Yaskawa INFORM job: DEMO_ROOF_SIDE_0625_3PAINT_31.JBI

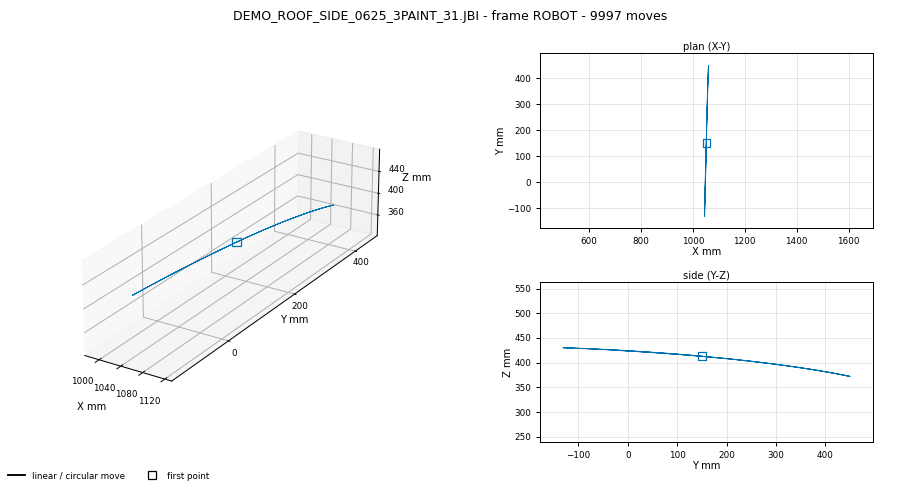
[picture p0: tool path of DEMO_ROOF_SIDE_0625_3PAINT_31.JBI in frame ROBOT, 9997 of 9997 moves have a stored position in this frame; points joined in program order, loops and branches not executed]
/JOB
//NAME DEMO_ROOF_SIDE_0625_3PAINT31
//POS
///NPOS 9997,0,0,0,0,0
///TOOL 0
///USER 0
///POSTYPE ROBOT
///RECTAN
///RCONF 1,0,0,0,0,0,0,0,0,0,0,0,0,0,0,0,0,0,0,0,0,0,0,0
C00000=1052.592,150.571,413.332,171.366,34.299,156.430
C00001=1052.586,150.322,413.353,171.364,34.297,156.430
C00002=1052.580,150.074,413.375,171.362,34.294,156.429
C00003=1052.574,149.824,413.397,171.360,34.291,156.429
C00004=1052.568,149.575,413.419,171.358,34.290,156.428
C00005=1052.563,149.326,413.440,171.357,34.287,156.428
C00006=1052.557,149.077,413.462,171.355,34.285,156.427
C00007=1052.550,148.828,413.484,171.353,34.283,156.427
C00008=1052.544,148.579,413.506,171.351,34.280,156.427
C00009=1052.538,148.331,413.527,171.349,34.278,156.426
C00010=1052.532,148.082,413.549,171.347,34.276,156.426
C00011=1052.526,147.832,413.571,171.345,34.273,156.425
C00012=1052.520,147.583,413.592,171.343,34.271,156.425
C00013=1052.515,147.334,413.614,171.341,34.269,156.425
C00014=1052.508,147.085,413.635,171.339,34.267,156.424
C00015=1052.502,146.836,413.657,171.337,34.264,156.424
C00016=1052.496,146.587,413.678,171.335,34.262,156.424
C00017=1052.490,146.339,413.700,171.334,34.260,156.423
C00018=1052.484,146.089,413.721,171.332,34.258,156.423
C00019=1052.478,145.840,413.743,171.330,34.255,156.422
C00020=1052.472,145.591,413.764,171.328,34.253,156.422
C00021=1052.466,145.342,413.786,171.326,34.251,156.422
C00022=1052.460,145.093,413.807,171.324,34.248,156.421
C00023=1052.454,144.844,413.829,171.322,34.246,156.421
C00024=1052.448,144.595,413.850,171.320,34.244,156.420
C00025=1052.442,144.346,413.872,171.318,34.242,156.420
C00026=1052.436,144.097,413.894,171.316,34.239,156.420
C00027=1052.431,143.849,413.915,171.314,34.237,156.419
C00028=1052.424,143.599,413.936,171.313,34.235,156.419
C00029=1052.418,143.350,413.958,171.311,34.233,156.418
C00030=1052.412,143.101,413.980,171.309,34.230,156.418
C00031=1052.406,142.852,414.001,171.307,34.228,156.418
C00032=1052.400,142.603,414.021,171.305,34.226,156.417
C00033=1052.393,142.318,414.046,171.303,34.223,156.417
C00034=1052.387,142.033,414.071,171.301,34.221,156.416
C00035=1052.380,141.747,414.095,171.298,34.218,156.416
C00036=1052.373,141.462,414.120,171.296,34.216,156.415
C00037=1052.367,141.213,414.142,171.294,34.213,156.415
C00038=1052.361,140.964,414.163,171.292,34.211,156.415
C00039=1052.356,140.715,414.184,171.291,34.209,156.414
C00040=1052.349,140.466,414.205,171.289,34.206,156.414
C00041=1052.343,140.217,414.226,171.287,34.204,156.413
C00042=1052.337,139.968,414.248,171.285,34.202,156.413
C00043=1052.331,139.719,414.269,171.284,34.200,156.413
C00044=1052.325,139.470,414.290,171.282,34.197,156.412
C00045=1052.319,139.221,414.311,171.280,34.195,156.412
C00046=1052.312,138.972,414.333,171.278,34.193,156.411
C00047=1052.307,138.723,414.354,171.275,34.191,156.411
C00048=1052.301,138.473,414.375,171.274,34.189,156.411
C00049=1052.295,138.225,414.396,171.272,34.187,156.410
C00050=1052.289,137.976,414.417,171.270,34.184,156.410
C00051=1052.282,137.727,414.439,171.268,34.182,156.410
C00052=1052.277,137.478,414.459,171.266,34.180,156.409
C00053=1052.271,137.228,414.481,171.265,34.178,156.409
C00054=1052.265,136.980,414.502,171.263,34.175,156.408
C00055=1052.259,136.730,414.522,171.261,34.173,156.408
C00056=1052.253,136.481,414.544,171.259,34.171,156.408
C00057=1052.246,136.233,414.565,171.258,34.169,156.407
C00058=1052.240,135.983,414.586,171.256,34.166,156.407
C00059=1052.235,135.735,414.607,171.254,34.164,156.406
C00060=1052.228,135.485,414.627,171.251,34.162,156.406
C00061=1052.222,135.236,414.649,171.249,34.160,156.406
C00062=1052.217,134.988,414.670,171.248,34.158,156.405
C00063=1052.210,134.738,414.691,171.246,34.155,156.405
C00064=1052.204,134.489,414.712,171.244,34.153,156.405
C00065=1052.199,134.240,414.733,171.242,34.151,156.404
C00066=1052.192,133.991,414.753,171.241,34.149,156.404
C00067=1052.186,133.742,414.774,171.239,34.146,156.403
C00068=1052.181,133.493,414.796,171.237,34.144,156.403
C00069=1052.174,133.244,414.817,171.235,34.142,156.403
C00070=1052.169,132.995,414.837,171.234,34.140,156.402
C00071=1052.163,132.746,414.859,171.232,34.137,156.402
C00072=1052.157,132.497,414.879,171.230,34.136,156.401
C00073=1052.150,132.248,414.900,171.227,34.133,156.401
C00074=1052.145,131.999,414.921,171.226,34.131,156.401
C00075=1052.138,131.750,414.942,171.224,34.129,156.400
C00076=1052.133,131.501,414.963,171.222,34.127,156.400
C00077=1052.126,131.251,414.983,171.220,34.125,156.400
C00078=1052.120,131.002,415.004,171.219,34.122,156.399
C00079=1052.114,130.753,415.024,171.217,34.120,156.399
C00080=1052.108,130.504,415.046,171.215,34.118,156.398
C00081=1052.102,130.255,415.066,171.213,34.116,156.398
C00082=1052.095,130.006,415.086,171.211,34.114,156.398
C00083=1052.090,129.757,415.108,171.210,34.111,156.397
C00084=1052.083,129.508,415.128,171.208,34.109,156.397
C00085=1052.077,129.259,415.149,171.206,34.107,156.397
C00086=1052.071,129.010,415.170,171.204,34.105,156.396
C00087=1052.065,128.761,415.190,171.203,34.103,156.396
C00088=1052.059,128.512,415.211,171.200,34.101,156.395
C00089=1052.053,128.263,415.231,171.198,34.098,156.395
C00090=1052.046,128.013,415.251,171.196,34.096,156.395
C00091=1052.041,127.765,415.273,171.195,34.095,156.394
C00092=1052.034,127.515,415.293,171.193,34.092,156.394
C00093=1052.028,127.266,415.313,171.191,34.090,156.394
C00094=1052.022,127.017,415.334,171.189,34.088,156.393
C00095=1052.016,126.768,415.355,171.188,34.086,156.393
C00096=1052.010,126.519,415.375,171.186,34.084,156.392
C00097=1052.003,126.234,415.399,171.184,34.081,156.392
C00098=1051.996,125.948,415.422,171.182,34.079,156.392
C00099=1051.988,125.663,415.446,171.180,34.076,156.391
C00100=1051.982,125.377,415.469,171.178,34.073,156.391
C00101=1051.975,125.129,415.489,171.176,34.071,156.390
C00102=1051.970,124.879,415.510,171.174,34.070,156.390
C00103=1051.964,124.630,415.530,171.172,34.067,156.390
C00104=1051.958,124.381,415.550,171.170,34.065,156.389
C00105=1051.952,124.131,415.571,171.168,34.063,156.389
C00106=1051.945,123.883,415.592,171.167,34.061,156.388
C00107=1051.939,123.634,415.612,171.165,34.059,156.388
C00108=1051.934,123.384,415.633,171.163,34.056,156.388
C00109=1051.928,123.136,415.653,171.162,34.054,156.387
C00110=1051.921,122.886,415.673,171.160,34.052,156.387
C00111=1051.916,122.637,415.694,171.158,34.050,156.387
C00112=1051.909,122.387,415.714,171.156,34.048,156.386
C00113=1051.903,122.139,415.735,171.155,34.046,156.386
C00114=1051.898,121.890,415.755,171.153,34.043,156.386
C00115=1051.891,121.641,415.776,171.151,34.041,156.385
C00116=1051.885,121.392,415.795,171.150,34.039,156.385
C00117=1051.880,121.143,415.816,171.147,34.037,156.384
C00118=1051.873,120.893,415.836,171.145,34.035,156.384
C00119=1051.867,120.644,415.856,171.143,34.032,156.384
C00120=1051.861,120.396,415.876,171.142,34.031,156.383
C00121=1051.855,120.146,415.897,171.140,34.028,156.383
C00122=1051.849,119.897,415.917,171.138,34.026,156.383
C00123=1051.843,119.648,415.937,171.137,34.024,156.382
C00124=1051.838,119.398,415.958,171.135,34.022,156.382
C00125=1051.832,119.149,415.978,171.133,34.020,156.381
C00126=1051.825,118.901,415.999,171.132,34.017,156.381
C00127=1051.819,118.652,416.019,171.130,34.015,156.381
C00128=1051.813,118.403,416.040,171.128,34.013,156.380
C00129=1051.807,118.154,416.059,171.126,34.011,156.380
C00130=1051.801,117.904,416.080,171.125,34.009,156.380
C00131=1051.796,117.655,416.100,171.123,34.006,156.379
C00132=1051.790,117.406,416.120,171.121,34.004,156.379
C00133=1051.784,117.157,416.140,171.119,34.002,156.378
C00134=1051.777,116.907,416.160,171.117,34.000,156.378
C00135=1051.772,116.658,416.180,171.115,33.998,156.378
C00136=1051.766,116.409,416.200,171.114,33.995,156.377
C00137=1051.760,116.161,416.220,171.112,33.993,156.377
C00138=1051.753,115.911,416.241,171.110,33.991,156.376
C00139=1051.748,115.662,416.261,171.109,33.989,156.376
C00140=1051.742,115.413,416.281,171.107,33.987,156.376
C00141=1051.736,115.164,416.301,171.105,33.984,156.375
C00142=1051.730,114.915,416.321,171.104,33.982,156.375
C00143=1051.724,114.666,416.342,171.102,33.980,156.375
C00144=1051.718,114.417,416.362,171.100,33.978,156.374
C00145=1051.713,114.168,416.381,171.099,33.975,156.374
C00146=1051.706,113.918,416.402,171.097,33.973,156.374
C00147=1051.700,113.669,416.422,171.095,33.971,156.373
C00148=1051.695,113.420,416.442,171.094,33.969,156.373
C00149=1051.689,113.171,416.462,171.092,33.967,156.372
C00150=1051.683,112.921,416.482,171.089,33.965,156.372
C00151=1051.677,112.672,416.502,171.088,33.963,156.372
C00152=1051.671,112.424,416.522,171.086,33.961,156.371
C00153=1051.665,112.175,416.542,171.084,33.959,156.371
C00154=1051.658,111.925,416.561,171.083,33.956,156.371
C00155=1051.652,111.676,416.581,171.081,33.954,156.370
C00156=1051.646,111.427,416.601,171.079,33.952,156.370
C00157=1051.640,111.178,416.621,171.078,33.950,156.369
C00158=1051.634,110.928,416.641,171.076,33.948,156.369
C00159=1051.627,110.679,416.660,171.074,33.946,156.369
C00160=1051.621,110.431,416.680,171.072,33.944,156.368
C00161=1051.615,110.145,416.703,171.071,33.941,156.368
C00162=1051.607,109.859,416.725,171.069,33.939,156.368
C00163=1051.601,109.574,416.748,171.067,33.936,156.367
C00164=1051.594,109.288,416.770,171.065,33.934,156.367
C00165=1051.588,109.039,416.790,171.063,33.932,156.366
C00166=1051.581,108.790,416.810,171.061,33.930,156.366
C00167=1051.575,108.540,416.830,171.059,33.928,156.366
C00168=1051.569,108.292,416.849,171.057,33.926,156.365
C00169=1051.563,108.042,416.868,171.055,33.923,156.365
C00170=1051.557,107.793,416.888,171.054,33.921,156.365
C00171=1051.550,107.544,416.909,171.052,33.919,156.364
C00172=1051.545,107.294,416.928,171.050,33.917,156.364
C00173=1051.539,107.046,416.948,171.049,33.915,156.364
C00174=1051.532,106.797,416.966,171.047,33.913,156.363
C00175=1051.526,106.548,416.986,171.045,33.911,156.363
C00176=1051.520,106.298,417.007,171.044,33.908,156.362
C00177=1051.514,106.049,417.026,171.042,33.906,156.362
C00178=1051.508,105.800,417.046,171.040,33.905,156.362
C00179=1051.502,105.551,417.065,171.039,33.903,156.361
C00180=1051.495,105.302,417.085,171.037,33.900,156.361
C00181=1051.490,105.053,417.104,171.035,33.898,156.361
C00182=1051.484,104.804,417.124,171.034,33.896,156.360
C00183=1051.478,104.554,417.143,171.032,33.894,156.360
C00184=1051.472,104.305,417.163,171.030,33.892,156.360
C00185=1051.466,104.055,417.183,171.029,33.890,156.359
C00186=1051.459,103.807,417.202,171.027,33.888,156.359
C00187=1051.453,103.557,417.221,171.025,33.885,156.359
C00188=1051.447,103.309,417.241,171.023,33.883,156.358
C00189=1051.442,103.059,417.260,171.021,33.881,156.358
C00190=1051.436,102.810,417.280,171.020,33.879,156.357
C00191=1051.429,102.561,417.299,171.018,33.877,156.357
C00192=1051.423,102.311,417.319,171.016,33.875,156.357
C00193=1051.417,102.062,417.339,171.015,33.872,156.356
C00194=1051.411,101.813,417.358,171.013,33.870,156.356
C00195=1051.405,101.564,417.378,171.011,33.868,156.356
C00196=1051.399,101.315,417.396,171.010,33.866,156.355
C00197=1051.393,101.066,417.416,171.008,33.864,156.355
C00198=1051.387,100.817,417.436,171.006,33.862,156.355
C00199=1051.382,100.567,417.455,171.005,33.860,156.354
C00200=1051.375,100.318,417.473,171.003,33.857,156.354
C00201=1051.369,100.069,417.493,171.001,33.856,156.353
C00202=1051.363,99.820,417.512,171.000,33.854,156.353
C00203=1051.356,99.570,417.532,170.998,33.852,156.353
C00204=1051.350,99.321,417.552,170.996,33.850,156.353
C00205=1051.344,99.072,417.570,170.995,33.847,156.352
C00206=1051.338,98.823,417.590,170.993,33.845,156.352
C00207=1051.332,98.574,417.609,170.991,33.843,156.351
C00208=1051.326,98.325,417.628,170.989,33.841,156.351
C00209=1051.319,98.076,417.647,170.987,33.839,156.351
C00210=1051.314,97.826,417.666,170.986,33.837,156.350
C00211=1051.307,97.578,417.685,170.984,33.835,156.350
C00212=1051.301,97.328,417.705,170.982,33.833,156.350
C00213=1051.296,97.079,417.724,170.981,33.831,156.349
C00214=1051.289,96.830,417.743,170.979,33.829,156.349
C00215=1051.284,96.580,417.762,170.977,33.826,156.349
C00216=1051.277,96.332,417.781,170.976,33.825,156.348
C00217=1051.271,96.082,417.801,170.974,33.823,156.348
C00218=1051.264,95.833,417.819,170.972,33.821,156.348
C00219=1051.258,95.583,417.839,170.971,33.818,156.347
C00220=1051.252,95.334,417.857,170.969,33.816,156.347
C00221=1051.246,95.085,417.877,170.968,33.814,156.347
C00222=1051.240,94.836,417.896,170.966,33.812,156.346
C00223=1051.234,94.587,417.915,170.964,33.810,156.346
C00224=1051.227,94.338,417.934,170.963,33.808,156.345
C00225=1051.221,94.053,417.956,170.961,33.806,156.345
C00226=1051.213,93.766,417.977,170.959,33.803,156.345
C00227=1051.207,93.481,417.999,170.957,33.801,156.344
C00228=1051.200,93.196,418.021,170.954,33.798,156.344
C00229=1051.194,92.946,418.040,170.953,33.796,156.343
C00230=1051.188,92.697,418.059,170.951,33.794,156.343
C00231=1051.182,92.448,418.078,170.949,33.792,156.343
C00232=1051.176,92.199,418.097,170.948,33.790,156.342
C00233=1051.170,91.950,418.116,170.946,33.788,156.342
C00234=1051.163,91.701,418.135,170.944,33.786,156.342
C00235=1051.158,91.451,418.154,170.943,33.784,156.341
C00236=1051.151,91.202,418.173,170.941,33.781,156.341
C00237=1051.146,90.953,418.192,170.939,33.779,156.341
C00238=1051.140,90.703,418.211,170.938,33.777,156.340
C00239=1051.134,90.454,418.230,170.936,33.775,156.340
C00240=1051.127,90.205,418.249,170.935,33.773,156.340
C00241=1051.121,89.955,418.268,170.933,33.771,156.339
C00242=1051.115,89.706,418.287,170.931,33.769,156.339
C00243=1051.109,89.457,418.305,170.930,33.767,156.339
C00244=1051.102,89.208,418.324,170.928,33.765,156.338
C00245=1051.096,88.959,418.343,170.926,33.763,156.338
C00246=1051.090,88.710,418.362,170.925,33.761,156.338
C00247=1051.084,88.460,418.380,170.923,33.759,156.337
C00248=1051.077,88.211,418.398,170.921,33.756,156.337
C00249=1051.072,87.961,418.418,170.920,33.755,156.337
C00250=1051.065,87.712,418.436,170.918,33.753,156.336
C00251=1051.059,87.463,418.455,170.917,33.751,156.336
C00252=1051.053,87.215,418.473,170.915,33.749,156.336
C00253=1051.047,86.965,418.492,170.913,33.747,156.335
C00254=1051.041,86.716,418.511,170.911,33.745,156.335
C00255=1051.035,86.467,418.530,170.909,33.742,156.335
C00256=1051.028,86.217,418.548,170.907,33.740,156.334
C00257=1051.022,85.968,418.566,170.906,33.738,156.334
C00258=1051.016,85.719,418.586,170.904,33.736,156.334
C00259=1051.010,85.469,418.604,170.903,33.734,156.333
C00260=1051.004,85.220,418.623,170.901,33.732,156.333
C00261=1050.997,84.971,418.641,170.899,33.730,156.333
C00262=1050.992,84.721,418.660,170.898,33.728,156.332
C00263=1050.986,84.473,418.678,170.896,33.726,156.332
C00264=1050.979,84.224,418.697,170.894,33.724,156.331
C00265=1050.973,83.975,418.716,170.893,33.722,156.331
C00266=1050.967,83.725,418.734,170.891,33.720,156.331
C00267=1050.961,83.475,418.753,170.890,33.718,156.331
C00268=1050.955,83.226,418.771,170.888,33.716,156.330
C00269=1050.948,82.977,418.790,170.886,33.714,156.330
C00270=1050.943,82.729,418.808,170.885,33.712,156.329
C00271=1050.937,82.479,418.827,170.883,33.710,156.329
C00272=1050.931,82.230,418.846,170.881,33.708,156.329
C00273=1050.924,81.980,418.864,170.880,33.705,156.328
C00274=1050.918,81.731,418.882,170.878,33.703,156.328
C00275=1050.912,81.482,418.901,170.877,33.701,156.328
C00276=1050.907,81.233,418.920,170.875,33.699,156.327
C00277=1050.900,80.984,418.938,170.873,33.697,156.327
C00278=1050.894,80.734,418.956,170.872,33.695,156.327
C00279=1050.888,80.485,418.975,170.870,33.693,156.326
C00280=1050.881,80.236,418.994,170.868,33.691,156.326
C00281=1050.876,79.987,419.011,170.866,33.689,156.326
C00282=1050.870,79.737,419.030,170.864,33.687,156.325
C00283=1050.864,79.488,419.049,170.863,33.685,156.325
C00284=1050.858,79.238,419.067,170.861,33.682,156.325
C00285=1050.851,78.989,419.086,170.859,33.680,156.324
C00286=1050.846,78.740,419.103,170.858,33.679,156.324
C00287=1050.839,78.491,419.122,170.856,33.677,156.324
C00288=1050.833,78.242,419.140,170.855,33.675,156.323
C00289=1050.826,77.956,419.162,170.853,33.672,156.323
C00290=1050.819,77.670,419.182,170.851,33.670,156.323
C00291=1050.812,77.384,419.203,170.849,33.667,156.322
C00292=1050.805,77.099,419.224,170.847,33.665,156.322
C00293=1050.798,76.850,419.243,170.845,33.663,156.321
C00294=1050.793,76.601,419.260,170.844,33.661,156.321
C00295=1050.786,76.352,419.279,170.842,33.659,156.321
C00296=1050.780,76.102,419.297,170.841,33.657,156.320
C00297=1050.774,75.853,419.315,170.839,33.655,156.320
C00298=1050.768,75.603,419.333,170.837,33.653,156.320
C00299=1050.762,75.354,419.352,170.836,33.651,156.319
C00300=1050.756,75.105,419.370,170.834,33.649,156.319
C00301=1050.749,74.856,419.388,170.832,33.647,156.319
C00302=1050.743,74.606,419.406,170.831,33.645,156.318
C00303=1050.737,74.357,419.424,170.829,33.643,156.318
C00304=1050.731,74.108,419.442,170.828,33.641,156.318
C00305=1050.725,73.859,419.461,170.826,33.639,156.317
C00306=1050.718,73.609,419.478,170.824,33.637,156.317
C00307=1050.713,73.360,419.496,170.823,33.635,156.317
C00308=1050.706,73.111,419.515,170.821,33.633,156.316
C00309=1050.700,72.861,419.532,170.820,33.631,156.316
C00310=1050.694,72.612,419.551,170.818,33.629,156.316
C00311=1050.688,72.363,419.569,170.816,33.626,156.315
C00312=1050.682,72.113,419.587,170.814,33.624,156.315
C00313=1050.676,71.864,419.605,170.812,33.622,156.315
C00314=1050.670,71.615,419.623,170.810,33.620,156.314
C00315=1050.664,71.366,419.641,170.809,33.619,156.314
C00316=1050.657,71.117,419.659,170.807,33.617,156.314
C00317=1050.651,70.867,419.677,170.806,33.615,156.313
C00318=1050.645,70.618,419.695,170.804,33.613,156.313
C00319=1050.639,70.369,419.713,170.802,33.611,156.313
C00320=1050.633,70.119,419.731,170.801,33.608,156.312
C00321=1050.627,69.871,419.749,170.799,33.606,156.312
C00322=1050.621,69.621,419.767,170.797,33.604,156.312
C00323=1050.614,69.371,419.784,170.796,33.602,156.311
C00324=1050.608,69.122,419.802,170.794,33.600,156.311
C00325=1050.602,68.873,419.821,170.793,33.598,156.311
C00326=1050.596,68.623,419.839,170.791,33.596,156.310
C00327=1050.590,68.374,419.856,170.789,33.594,156.310
C00328=1050.583,68.125,419.874,170.788,33.592,156.310
C00329=1050.577,67.876,419.892,170.786,33.590,156.309
C00330=1050.571,67.627,419.910,170.784,33.588,156.309
C00331=1050.565,67.377,419.928,170.783,33.586,156.309
C00332=1050.558,67.128,419.945,170.781,33.584,156.309
C00333=1050.553,66.879,419.963,170.780,33.582,156.308
C00334=1050.546,66.630,419.981,170.778,33.580,156.308
C00335=1050.540,66.380,419.999,170.776,33.578,156.307
C00336=1050.534,66.131,420.016,170.775,33.576,156.307
C00337=1050.528,65.881,420.034,170.773,33.574,156.307
C00338=1050.521,65.632,420.051,170.771,33.572,156.306
C00339=1050.515,65.383,420.070,170.770,33.570,156.306
C00340=1050.509,65.134,420.088,170.768,33.568,156.306
C00341=1050.503,64.884,420.106,170.767,33.566,156.306
C00342=1050.497,64.635,420.123,170.765,33.564,156.305
C00343=1050.491,64.386,420.140,170.763,33.562,156.305
C00344=1050.485,64.136,420.158,170.762,33.560,156.305
C00345=1050.478,63.887,420.175,170.760,33.558,156.304
C00346=1050.472,63.637,420.193,170.758,33.556,156.304
C00347=1050.466,63.389,420.210,170.757,33.554,156.304
C00348=1050.459,63.140,420.228,170.755,33.552,156.303
C00349=1050.453,62.890,420.246,170.753,33.550,156.303
C00350=1050.446,62.641,420.263,170.752,33.548,156.303
C00351=1050.440,62.392,420.281,170.750,33.546,156.302
C00352=1050.433,62.142,420.298,170.749,33.545,156.302
C00353=1050.426,61.856,420.318,170.746,33.543,156.302
C00354=1050.419,61.570,420.338,170.744,33.541,156.301
C00355=1050.412,61.284,420.358,170.742,33.538,156.301
C00356=1050.405,60.999,420.378,170.740,33.536,156.301
C00357=1050.399,60.749,420.396,170.738,33.534,156.300
C00358=1050.392,60.500,420.413,170.737,33.532,156.300
C00359=1050.386,60.251,420.431,170.735,33.530,156.300
C00360=1050.379,60.001,420.448,170.733,33.528,156.299
C00361=1050.374,59.752,420.465,170.732,33.526,156.299
C00362=1050.367,59.503,420.483,170.730,33.524,156.299
C00363=1050.361,59.254,420.500,170.729,33.522,156.298
C00364=1050.355,59.004,420.518,170.727,33.520,156.298
C00365=1050.348,58.755,420.535,170.725,33.518,156.298
C00366=1050.342,58.506,420.553,170.724,33.516,156.297
C00367=1050.335,58.256,420.570,170.722,33.514,156.297
C00368=1050.329,58.008,420.587,170.720,33.513,156.297
C00369=1050.323,57.758,420.605,170.719,33.511,156.297
C00370=1050.317,57.509,420.622,170.717,33.509,156.296
C00371=1050.311,57.259,420.639,170.715,33.507,156.296
C00372=1050.305,57.010,420.656,170.714,33.505,156.296
C00373=1050.298,56.761,420.673,170.712,33.503,156.295
C00374=1050.292,56.511,420.691,170.711,33.501,156.295
C00375=1050.285,56.262,420.708,170.709,33.499,156.295
C00376=1050.279,56.012,420.726,170.707,33.497,156.294
C00377=1050.273,55.763,420.742,170.706,33.495,156.294
C00378=1050.267,55.514,420.760,170.704,33.493,156.294
C00379=1050.261,55.264,420.777,170.702,33.491,156.293
C00380=1050.254,55.015,420.795,170.701,33.489,156.293
C00381=1050.249,54.766,420.812,170.699,33.487,156.293
C00382=1050.242,54.516,420.829,170.697,33.485,156.293
C00383=1050.236,54.267,420.846,170.696,33.483,156.292
C00384=1050.230,54.017,420.864,170.694,33.481,156.292
C00385=1050.223,53.769,420.881,170.692,33.479,156.292
C00386=1050.217,53.519,420.898,170.691,33.477,156.291
C00387=1050.211,53.270,420.915,170.689,33.475,156.291
C00388=1050.205,53.020,420.932,170.688,33.473,156.291
C00389=1050.199,52.771,420.950,170.686,33.471,156.290
C00390=1050.193,52.522,420.967,170.684,33.469,156.290
C00391=1050.186,52.272,420.983,170.683,33.467,156.290
C00392=1050.181,52.023,421.001,170.681,33.465,156.289
C00393=1050.174,51.774,421.018,170.679,33.463,156.289
C00394=1050.168,51.525,421.035,170.678,33.462,156.289
C00395=1050.162,51.275,421.053,170.676,33.459,156.288
C00396=1050.155,51.026,421.069,170.674,33.457,156.288
C00397=1050.149,50.776,421.086,170.673,33.456,156.288
C00398=1050.143,50.527,421.104,170.671,33.454,156.287
C00399=1050.137,50.278,421.121,170.670,33.452,156.287
C00400=1050.131,50.028,421.137,170.668,33.450,156.287
C00401=1050.125,49.779,421.155,170.666,33.448,156.287
C00402=1050.118,49.530,421.172,170.665,33.446,156.286
C00403=1050.113,49.280,421.189,170.663,33.444,156.286
C00404=1050.107,49.031,421.206,170.661,33.442,156.286
C00405=1050.100,48.782,421.223,170.660,33.440,156.285
C00406=1050.095,48.532,421.240,170.658,33.438,156.285
C00407=1050.088,48.283,421.258,170.657,33.436,156.285
C00408=1050.082,48.034,421.274,170.655,33.434,156.284
C00409=1050.076,47.785,421.291,170.653,33.432,156.284
C00410=1050.069,47.535,421.309,170.652,33.430,156.284
C00411=1050.064,47.286,421.325,170.650,33.428,156.283
C00412=1050.057,47.037,421.342,170.648,33.426,156.283
C00413=1050.051,46.787,421.359,170.647,33.424,156.283
C00414=1050.045,46.538,421.376,170.644,33.422,156.282
C00415=1050.039,46.289,421.392,170.642,33.420,156.282
C00416=1050.033,46.039,421.410,170.641,33.418,156.282
C00417=1050.026,45.752,421.430,170.639,33.415,156.281
C00418=1050.019,45.467,421.449,170.637,33.413,156.281
C00419=1050.012,45.180,421.468,170.635,33.411,156.281
C00420=1050.005,44.894,421.488,170.633,33.409,156.280
C00421=1049.999,44.645,421.504,170.632,33.407,156.280
C00422=1049.993,44.396,421.521,170.630,33.405,156.280
C00423=1049.988,44.146,421.538,170.628,33.403,156.279
C00424=1049.981,43.897,421.555,170.627,33.401,156.279
C00425=1049.975,43.648,421.572,170.625,33.399,156.279
C00426=1049.969,43.399,421.589,170.623,33.397,156.278
C00427=1049.963,43.149,421.606,170.622,33.395,156.278
C00428=1049.957,42.900,421.623,170.620,33.393,156.278
C00429=1049.951,42.650,421.639,170.619,33.391,156.277
C00430=1049.944,42.400,421.656,170.617,33.389,156.277
C00431=1049.938,42.152,421.673,170.615,33.387,156.277
C00432=1049.932,41.902,421.689,170.614,33.386,156.277
C00433=1049.925,41.652,421.706,170.612,33.384,156.276
C00434=1049.919,41.404,421.723,170.610,33.382,156.276
C00435=1049.913,41.154,421.739,170.609,33.380,156.276
C00436=1049.906,40.905,421.756,170.607,33.378,156.275
C00437=1049.900,40.655,421.772,170.605,33.376,156.275
C00438=1049.894,40.406,421.789,170.604,33.374,156.275
C00439=1049.888,40.157,421.806,170.602,33.372,156.274
C00440=1049.882,39.907,421.822,170.600,33.370,156.274
C00441=1049.876,39.658,421.839,170.599,33.368,156.274
C00442=1049.870,39.409,421.855,170.597,33.366,156.273
C00443=1049.863,39.159,421.872,170.595,33.364,156.273
C00444=1049.858,38.910,421.889,170.594,33.362,156.273
C00445=1049.852,38.660,421.905,170.592,33.360,156.273
C00446=1049.845,38.411,421.922,170.590,33.358,156.272
C00447=1049.839,38.161,421.939,170.589,33.356,156.272
C00448=1049.833,37.912,421.955,170.587,33.354,156.272
C00449=1049.827,37.663,421.971,170.585,33.352,156.271
C00450=1049.821,37.414,421.988,170.584,33.350,156.271
C00451=1049.813,37.164,422.004,170.582,33.348,156.271
C00452=1049.807,36.915,422.021,170.580,33.347,156.271
C00453=1049.801,36.666,422.037,170.579,33.345,156.270
C00454=1049.795,36.415,422.054,170.577,33.343,156.270
C00455=1049.789,36.166,422.070,170.575,33.341,156.270
C00456=1049.783,35.917,422.087,170.574,33.339,156.269
C00457=1049.777,35.668,422.103,170.572,33.338,156.269
C00458=1049.769,35.418,422.119,170.570,33.336,156.269
C00459=1049.764,35.169,422.135,170.569,33.334,156.268
C00460=1049.758,34.920,422.152,170.567,33.332,156.268
C00461=1049.752,34.670,422.168,170.565,33.330,156.268
C00462=1049.745,34.421,422.185,170.564,33.328,156.268
C00463=1049.739,34.171,422.201,170.562,33.326,156.267
C00464=1049.732,33.922,422.217,170.560,33.324,156.267
C00465=1049.726,33.673,422.233,170.558,33.322,156.267
C00466=1049.720,33.424,422.250,170.557,33.320,156.266
C00467=1049.714,33.174,422.266,170.555,33.318,156.266
C00468=1049.708,32.924,422.282,170.553,33.317,156.266
C00469=1049.701,32.675,422.298,170.552,33.315,156.266
C00470=1049.695,32.426,422.314,170.550,33.313,156.265
C00471=1049.689,32.177,422.331,170.548,33.311,156.265
C00472=1049.683,31.927,422.347,170.547,33.309,156.265
C00473=1049.677,31.677,422.364,170.545,33.307,156.264
C00474=1049.671,31.428,422.380,170.543,33.306,156.264
C00475=1049.664,31.179,422.395,170.542,33.304,156.264
C00476=1049.658,30.929,422.412,170.540,33.302,156.264
C00477=1049.651,30.679,422.428,170.538,33.300,156.263
C00478=1049.646,30.430,422.445,170.537,33.298,156.263
C00479=1049.640,30.181,422.461,170.535,33.296,156.263
C00480=1049.633,29.932,422.476,170.533,33.294,156.262
C00481=1049.625,29.645,422.495,170.531,33.292,156.262
C00482=1049.619,29.360,422.514,170.529,33.290,156.262
C00483=1049.612,29.073,422.533,170.527,33.288,156.261
C00484=1049.605,28.787,422.551,170.526,33.286,156.261
C00485=1049.599,28.538,422.568,170.524,33.284,156.261
C00486=1049.592,28.289,422.583,170.522,33.282,156.260
C00487=1049.586,28.039,422.599,170.520,33.280,156.260
C00488=1049.580,27.790,422.616,170.519,33.278,156.260
C00489=1049.573,27.540,422.631,170.517,33.276,156.260
C00490=1049.567,27.290,422.647,170.515,33.274,156.259
C00491=1049.560,27.041,422.663,170.514,33.272,156.259
C00492=1049.555,26.792,422.679,170.512,33.271,156.259
C00493=1049.549,26.543,422.695,170.510,33.269,156.258
C00494=1049.542,26.294,422.711,170.509,33.267,156.258
C00495=1049.536,26.044,422.727,170.507,33.265,156.258
C00496=1049.530,25.794,422.743,170.505,33.263,156.258
C00497=1049.523,25.545,422.759,170.503,33.261,156.257
C00498=1049.517,25.295,422.775,170.502,33.259,156.257
C00499=1049.510,25.046,422.791,170.500,33.257,156.257
C00500=1049.504,24.797,422.807,170.498,33.256,156.257
C00501=1049.498,24.548,422.823,170.497,33.254,156.256
C00502=1049.492,24.298,422.838,170.495,33.252,156.256
C00503=1049.486,24.048,422.855,170.493,33.251,156.256
C00504=1049.479,23.799,422.870,170.491,33.249,156.255
C00505=1049.473,23.550,422.886,170.490,33.247,156.255
C00506=1049.466,23.300,422.902,170.488,33.245,156.255
C00507=1049.461,23.050,422.918,170.486,33.243,156.255
C00508=1049.454,22.801,422.934,170.485,33.241,156.254
C00509=1049.448,22.552,422.950,170.483,33.239,156.254
C00510=1049.442,22.302,422.965,170.481,33.237,156.254
C00511=1049.436,22.053,422.981,170.480,33.236,156.253
C00512=1049.430,21.804,422.997,170.478,33.234,156.253
C00513=1049.423,21.554,423.012,170.476,33.232,156.253
C00514=1049.417,21.305,423.029,170.474,33.230,156.253
C00515=1049.411,21.056,423.044,170.473,33.228,156.252
C00516=1049.405,20.806,423.060,170.471,33.226,156.252
C00517=1049.398,20.557,423.075,170.469,33.224,156.252
C00518=1049.392,20.307,423.092,170.468,33.223,156.252
C00519=1049.386,20.058,423.107,170.466,33.221,156.251
C00520=1049.380,19.808,423.123,170.464,33.219,156.251
C00521=1049.373,19.559,423.139,170.462,33.218,156.251
C00522=1049.368,19.309,423.154,170.461,33.216,156.250
C00523=1049.361,19.060,423.170,170.459,33.214,156.250
C00524=1049.355,18.811,423.186,170.457,33.212,156.250
C00525=1049.349,18.561,423.201,170.455,33.210,156.250
C00526=1049.342,18.312,423.217,170.454,33.208,156.249
C00527=1049.336,18.062,423.232,170.452,33.207,156.249
C00528=1049.330,17.813,423.248,170.450,33.205,156.249
C00529=1049.324,17.563,423.263,170.449,33.203,156.248
C00530=1049.317,17.314,423.279,170.447,33.201,156.248
C00531=1049.311,17.064,423.294,170.445,33.199,156.248
C00532=1049.305,16.815,423.310,170.443,33.197,156.248
C00533=1049.298,16.566,423.326,170.442,33.196,156.247
C00534=1049.293,16.316,423.341,170.440,33.194,156.247
C00535=1049.286,16.067,423.357,170.438,33.192,156.247
C00536=1049.280,15.817,423.372,170.436,33.191,156.247
C00537=1049.274,15.568,423.388,170.435,33.189,156.246
C00538=1049.267,15.318,423.403,170.433,33.187,156.246
C00539=1049.261,15.069,423.420,170.431,33.185,156.246
C00540=1049.255,14.819,423.435,170.429,33.183,156.246
C00541=1049.248,14.570,423.450,170.428,33.181,156.245
C00542=1049.243,14.320,423.466,170.426,33.180,156.245
C00543=1049.236,14.071,423.481,170.424,33.178,156.245
C00544=1049.229,13.822,423.496,170.422,33.176,156.244
C00545=1049.224,13.605,423.509,170.421,33.174,156.244
C00546=1049.218,13.389,423.523,170.419,33.173,156.244
C00547=1049.213,13.173,423.536,170.418,33.172,156.244
C00548=1049.208,12.957,423.550,170.416,33.170,156.244
C00549=1049.202,12.740,423.563,170.415,33.168,156.243
C00550=1049.196,12.524,423.576,170.413,33.167,156.243
C00551=1049.191,12.307,423.589,170.412,33.166,156.243
C00552=1049.185,12.091,423.603,170.410,33.164,156.243
C00553=1049.179,11.842,423.618,170.408,33.162,156.242
C00554=1049.173,11.592,423.633,170.407,33.161,156.242
C00555=1049.166,11.343,423.648,170.405,33.159,156.242
C00556=1049.160,11.093,423.664,170.403,33.157,156.242
C00557=1049.154,10.843,423.679,170.401,33.155,156.241
C00558=1049.147,10.594,423.694,170.400,33.154,156.241
C00559=1049.141,10.345,423.709,170.398,33.152,156.241
C00560=1049.135,10.096,423.724,170.397,33.150,156.241
C00561=1049.129,9.846,423.739,170.395,33.148,156.240
C00562=1049.122,9.597,423.755,170.394,33.147,156.240
C00563=1049.116,9.347,423.770,170.392,33.145,156.240
C00564=1049.110,9.097,423.785,170.390,33.143,156.240
C00565=1049.103,8.848,423.801,170.388,33.142,156.239
C00566=1049.097,8.599,423.816,170.386,33.140,156.239
C00567=1049.090,8.349,423.831,170.385,33.138,156.239
C00568=1049.084,8.099,423.846,170.383,33.136,156.239
C00569=1049.077,7.850,423.861,170.381,33.135,156.238
C00570=1049.072,7.601,423.876,170.379,33.133,156.238
C00571=1049.066,7.351,423.891,170.378,33.131,156.238
C00572=1049.060,7.102,423.906,170.376,33.129,156.238
C00573=1049.051,6.751,423.928,170.373,33.127,156.237
C00574=1049.042,6.399,423.949,170.371,33.125,156.237
C00575=1049.033,6.049,423.970,170.368,33.122,156.237
C00576=1049.024,5.697,423.991,170.366,33.120,156.236
C00577=1049.018,5.447,424.006,170.364,33.118,156.236
C00578=1049.011,5.198,424.022,170.362,33.116,156.236
C00579=1049.005,4.949,424.037,170.360,33.114,156.235
C00580=1048.999,4.699,424.052,170.359,33.113,156.235
C00581=1048.993,4.450,424.066,170.357,33.111,156.235
C00582=1048.986,4.200,424.081,170.355,33.109,156.235
C00583=1048.980,3.951,424.096,170.353,33.107,156.234
C00584=1048.974,3.701,424.111,170.352,33.106,156.234
C00585=1048.967,3.451,424.126,170.350,33.104,156.234
C00586=1048.961,3.203,424.141,170.348,33.103,156.234
C00587=1048.955,2.953,424.157,170.346,33.101,156.233
C00588=1048.949,2.703,424.172,170.344,33.099,156.233
C00589=1048.943,2.454,424.187,170.343,33.097,156.233
C00590=1048.937,2.205,424.201,170.341,33.096,156.233
C00591=1048.931,1.955,424.216,170.339,33.094,156.232
C00592=1048.924,1.706,424.231,170.337,33.092,156.232
C00593=1048.918,1.456,424.246,170.335,33.090,156.232
C00594=1048.912,1.207,424.261,170.334,33.088,156.232
C00595=1048.906,0.957,424.276,170.332,33.087,156.231
C00596=1048.899,0.708,424.291,170.330,33.085,156.231
C00597=1048.893,0.458,424.306,170.328,33.083,156.231
C00598=1048.887,0.209,424.320,170.326,33.081,156.231
C00599=1048.881,-0.041,424.335,170.325,33.080,156.230
C00600=1048.874,-0.290,424.350,170.323,33.078,156.230
C00601=1048.869,-0.539,424.365,170.321,33.077,156.230
C00602=1048.862,-0.789,424.380,170.319,33.075,156.230
C00603=1048.857,-1.039,424.395,170.317,33.073,156.229
C00604=1048.850,-1.289,424.410,170.316,33.071,156.229
C00605=1048.844,-1.537,424.425,170.314,33.070,156.229
C00606=1048.838,-1.787,424.440,170.312,33.068,156.229
C00607=1048.832,-2.037,424.454,170.310,33.066,156.228
C00608=1048.826,-2.286,424.469,170.308,33.064,156.228
C00609=1048.819,-2.569,424.485,170.306,33.062,156.228
C00610=1048.811,-2.852,424.502,170.304,33.060,156.228
C00611=1048.805,-3.135,424.518,170.302,33.059,156.227
C00612=1048.797,-3.418,424.536,170.300,33.057,156.227
C00613=1048.791,-3.667,424.550,170.298,33.055,156.227
C00614=1048.785,-3.918,424.565,170.297,33.053,156.227
C00615=1048.779,-4.167,424.579,170.295,33.052,156.226
C00616=1048.772,-4.416,424.594,170.293,33.050,156.226
C00617=1048.766,-4.666,424.609,170.291,33.048,156.226
C00618=1048.760,-4.915,424.623,170.289,33.047,156.226
C00619=1048.754,-5.164,424.638,170.287,33.045,156.225
C00620=1048.747,-5.414,424.652,170.286,33.044,156.225
C00621=1048.741,-5.663,424.666,170.284,33.042,156.225
C00622=1048.735,-5.913,424.681,170.283,33.040,156.225
C00623=1048.728,-6.162,424.696,170.281,33.039,156.225
C00624=1048.721,-6.412,424.710,170.279,33.037,156.224
C00625=1048.716,-6.661,424.724,170.277,33.035,156.224
C00626=1048.709,-6.911,424.739,170.276,33.034,156.224
C00627=1048.702,-7.160,424.754,170.274,33.032,156.224
C00628=1048.697,-7.410,424.768,170.272,33.030,156.223
C00629=1048.690,-7.660,424.783,170.270,33.029,156.223
C00630=1048.684,-7.909,424.797,170.268,33.028,156.223
C00631=1048.678,-8.158,424.811,170.266,33.025,156.223
C00632=1048.671,-8.408,424.826,170.264,33.024,156.222
C00633=1048.665,-8.657,424.840,170.263,33.023,156.222
C00634=1048.659,-8.907,424.854,170.261,33.021,156.222
C00635=1048.652,-9.157,424.869,170.259,33.019,156.222
C00636=1048.646,-9.406,424.883,170.257,33.018,156.222
C00637=1048.640,-9.656,424.898,170.255,33.016,156.221
C00638=1048.634,-9.905,424.912,170.253,33.014,156.221
C00639=1048.628,-10.154,424.927,170.252,33.013,156.221
C00640=1048.621,-10.405,424.941,170.250,33.012,156.221
C00641=1048.615,-10.653,424.955,170.248,33.009,156.220
C00642=1048.609,-10.903,424.969,170.246,33.008,156.220
C00643=1048.603,-11.152,424.984,170.244,33.007,156.220
C00644=1048.596,-11.402,424.998,170.242,33.005,156.220
C00645=1048.590,-11.652,425.012,170.240,33.003,156.220
C00646=1048.584,-11.901,425.027,170.239,33.002,156.219
C00647=1048.577,-12.151,425.040,170.237,33.000,156.219
C00648=1048.571,-12.400,425.055,170.235,32.998,156.219
C00649=1048.565,-12.650,425.069,170.233,32.997,156.219
C00650=1048.559,-12.899,425.083,170.231,32.995,156.218
C00651=1048.552,-13.148,425.098,170.229,32.993,156.218
C00652=1048.547,-13.398,425.112,170.227,32.992,156.218
C00653=1048.541,-13.648,425.127,170.225,32.991,156.218
C00654=1048.534,-13.897,425.140,170.224,32.989,156.218
C00655=1048.528,-14.147,425.155,170.222,32.987,156.217
C00656=1048.522,-14.396,425.168,170.220,32.986,156.217
C00657=1048.515,-14.646,425.183,170.218,32.984,156.217
C00658=1048.509,-14.896,425.198,170.216,32.982,156.217
C00659=1048.503,-15.144,425.212,170.214,32.981,156.216
C00660=1048.497,-15.395,425.226,170.212,32.979,156.216
C00661=1048.491,-15.644,425.239,170.210,32.977,156.216
C00662=1048.484,-15.894,425.254,170.209,32.976,156.216
C00663=1048.478,-16.143,425.267,170.207,32.975,156.216
C00664=1048.472,-16.393,425.282,170.205,32.973,156.215
C00665=1048.465,-16.642,425.296,170.203,32.972,156.215
C00666=1048.459,-16.892,425.310,170.202,32.970,156.215
C00667=1048.453,-17.141,425.324,170.200,32.968,156.215
C00668=1048.447,-17.391,425.338,170.198,32.967,156.215
C00669=1048.440,-17.640,425.352,170.196,32.965,156.214
C00670=1048.433,-17.890,425.366,170.194,32.964,156.214
C00671=1048.428,-18.139,425.379,170.193,32.962,156.214
C00672=1048.421,-18.389,425.394,170.191,32.961,156.214
C00673=1048.414,-18.670,425.409,170.188,32.959,156.214
C00674=1048.407,-18.951,425.425,170.186,32.957,156.213
C00675=1048.400,-19.233,425.441,170.184,32.955,156.213
C00676=1048.393,-19.514,425.456,170.182,32.954,156.213
C00677=1048.387,-19.764,425.470,170.180,32.953,156.213
C00678=1048.380,-20.013,425.485,170.178,32.951,156.213
C00679=1048.374,-20.263,425.498,170.176,32.950,156.212
C00680=1048.368,-20.513,425.512,170.174,32.948,156.212
C00681=1048.362,-20.762,425.525,170.172,32.946,156.212
C00682=1048.355,-21.011,425.540,170.171,32.945,156.212
C00683=1048.349,-21.261,425.554,170.169,32.943,156.211
C00684=1048.342,-21.511,425.567,170.167,32.942,156.211
C00685=1048.337,-21.761,425.581,170.165,32.941,156.211
C00686=1048.330,-22.009,425.595,170.163,32.939,156.211
C00687=1048.323,-22.259,425.609,170.161,32.937,156.211
C00688=1048.318,-22.509,425.623,170.159,32.936,156.210
C00689=1048.311,-22.759,425.636,170.157,32.934,156.210
C00690=1048.306,-23.008,425.650,170.155,32.933,156.210
C00691=1048.299,-23.257,425.664,170.153,32.931,156.210
C00692=1048.292,-23.507,425.678,170.151,32.930,156.210
C00693=1048.287,-23.756,425.692,170.149,32.928,156.210
C00694=1048.280,-24.006,425.705,170.148,32.927,156.209
C00695=1048.274,-24.256,425.719,170.146,32.925,156.209
C00696=1048.268,-24.505,425.732,170.144,32.924,156.209
C00697=1048.261,-24.755,425.747,170.142,32.922,156.209
C00698=1048.256,-25.004,425.761,170.140,32.921,156.208
C00699=1048.250,-25.253,425.774,170.138,32.919,156.208
C00700=1048.243,-25.503,425.788,170.136,32.918,156.208
C00701=1048.237,-25.753,425.801,170.134,32.916,156.208
C00702=1048.231,-26.002,425.815,170.133,32.915,156.208
C00703=1048.224,-26.252,425.828,170.131,32.913,156.208
C00704=1048.219,-26.502,425.842,170.129,32.912,156.207
C00705=1048.213,-26.751,425.855,170.127,32.910,156.207
C00706=1048.205,-27.000,425.870,170.125,32.909,156.207
C00707=1048.200,-27.250,425.884,170.123,32.907,156.207
C00708=1048.193,-27.500,425.897,170.121,32.906,156.207
C00709=1048.187,-27.749,425.911,170.120,32.904,156.206
C00710=1048.181,-27.998,425.924,170.118,32.903,156.206
C00711=1048.174,-28.248,425.937,170.116,32.902,156.206
C00712=1048.168,-28.498,425.951,170.114,32.901,156.206
C00713=1048.161,-28.747,425.964,170.112,32.899,156.206
C00714=1048.155,-28.997,425.978,170.110,32.898,156.206
C00715=1048.149,-29.247,425.991,170.108,32.896,156.205
C00716=1048.143,-29.496,426.004,170.106,32.895,156.205
C00717=1048.136,-29.746,426.018,170.104,32.893,156.205
C00718=1048.130,-29.996,426.031,170.102,32.892,156.205
C00719=1048.124,-30.245,426.044,170.100,32.890,156.205
C00720=1048.117,-30.495,426.058,170.098,32.889,156.204
C00721=1048.111,-30.744,426.071,170.096,32.888,156.204
C00722=1048.105,-30.993,426.084,170.094,32.886,156.204
C00723=1048.099,-31.244,426.099,170.092,32.885,156.204
C00724=1048.092,-31.493,426.112,170.090,32.883,156.204
C00725=1048.086,-31.742,426.125,170.088,32.882,156.203
C00726=1048.080,-31.991,426.138,170.086,32.880,156.203
C00727=1048.074,-32.242,426.151,170.084,32.880,156.203
C00728=1048.067,-32.491,426.165,170.082,32.878,156.203
C00729=1048.061,-32.741,426.178,170.080,32.877,156.203
C00730=1048.055,-32.990,426.191,170.078,32.875,156.203
C00731=1048.048,-33.240,426.205,170.076,32.874,156.203
C00732=1048.042,-33.489,426.218,170.074,32.872,156.202
C00733=1048.036,-33.738,426.231,170.072,32.871,156.202
C00734=1048.030,-33.989,426.244,170.071,32.869,156.202
C00735=1048.024,-34.238,426.258,170.069,32.868,156.202
C00736=1048.017,-34.488,426.271,170.067,32.867,156.202
C00737=1048.010,-34.768,426.286,170.065,32.865,156.201
C00738=1048.003,-35.049,426.301,170.063,32.864,156.201
C00739=1047.997,-35.330,426.316,170.061,32.862,156.201
C00740=1047.990,-35.610,426.331,170.058,32.861,156.201
C00741=1047.983,-35.859,426.344,170.056,32.859,156.201
C00742=1047.977,-36.110,426.357,170.054,32.858,156.201
C00743=1047.971,-36.359,426.370,170.053,32.856,156.200
C00744=1047.964,-36.608,426.383,170.051,32.855,156.200
C00745=1047.958,-36.857,426.397,170.049,32.854,156.200
C00746=1047.952,-37.107,426.409,170.047,32.852,156.200
C00747=1047.946,-37.357,426.423,170.045,32.851,156.200
C00748=1047.939,-37.606,426.436,170.043,32.850,156.200
C00749=1047.933,-37.856,426.449,170.041,32.848,156.199
C00750=1047.927,-38.106,426.462,170.039,32.847,156.199
C00751=1047.921,-38.355,426.475,170.037,32.845,156.199
C00752=1047.915,-38.605,426.488,170.035,32.844,156.199
C00753=1047.909,-38.854,426.501,170.033,32.843,156.199
C00754=1047.902,-39.104,426.515,170.031,32.842,156.199
C00755=1047.896,-39.354,426.527,170.029,32.840,156.198
C00756=1047.890,-39.603,426.541,170.027,32.839,156.198
C00757=1047.884,-39.852,426.554,170.024,32.837,156.198
C00758=1047.877,-40.102,426.566,170.022,32.837,156.198
C00759=1047.871,-40.351,426.579,170.020,32.835,156.198
C00760=1047.864,-40.602,426.592,170.018,32.834,156.198
C00761=1047.858,-40.851,426.605,170.016,32.832,156.197
C00762=1047.852,-41.101,426.618,170.014,32.831,156.197
C00763=1047.846,-41.350,426.631,170.013,32.830,156.197
C00764=1047.839,-41.600,426.643,170.011,32.828,156.197
C00765=1047.833,-41.849,426.656,170.009,32.828,156.197
C00766=1047.827,-42.098,426.670,170.007,32.826,156.197
C00767=1047.820,-42.349,426.682,170.005,32.825,156.197
C00768=1047.814,-42.598,426.696,170.003,32.823,156.196
C00769=1047.808,-42.848,426.708,170.001,32.822,156.196
C00770=1047.801,-43.097,426.721,169.999,32.821,156.196
C00771=1047.795,-43.347,426.734,169.997,32.820,156.196
C00772=1047.789,-43.596,426.747,169.995,32.819,156.196
C00773=1047.783,-43.846,426.759,169.993,32.817,156.196
C00774=1047.777,-44.096,426.771,169.991,32.816,156.195
C00775=1047.770,-44.345,426.785,169.989,32.815,156.195
C00776=1047.765,-44.595,426.797,169.987,32.814,156.195
C00777=1047.758,-44.845,426.811,169.985,32.812,156.195
C00778=1047.752,-45.095,426.823,169.983,32.811,156.195
C00779=1047.745,-45.344,426.836,169.981,32.810,156.195
C00780=1047.739,-45.593,426.849,169.979,32.808,156.195
C00781=1047.733,-45.843,426.861,169.977,32.808,156.195
C00782=1047.727,-46.093,426.874,169.975,32.806,156.194
C00783=1047.721,-46.342,426.887,169.973,32.805,156.194
C00784=1047.714,-46.591,426.900,169.971,32.803,156.194
C00785=1047.708,-46.841,426.912,169.969,32.802,156.194
C00786=1047.702,-47.091,426.925,169.967,32.801,156.194
C00787=1047.696,-47.340,426.938,169.964,32.800,156.194
C00788=1047.689,-47.590,426.950,169.962,32.799,156.194
C00789=1047.683,-47.840,426.963,169.960,32.797,156.193
C00790=1047.677,-48.089,426.976,169.959,32.796,156.193
C00791=1047.671,-48.339,426.988,169.957,32.795,156.193
C00792=1047.665,-48.589,427.000,169.955,32.793,156.193
C00793=1047.658,-48.838,427.014,169.953,32.793,156.193
C00794=1047.652,-49.088,427.026,169.951,32.791,156.193
C00795=1047.647,-49.338,427.039,169.949,32.790,156.193
C00796=1047.640,-49.587,427.051,169.947,32.789,156.192
C00797=1047.634,-49.837,427.064,169.945,32.787,156.192
C00798=1047.628,-50.086,427.076,169.943,32.786,156.192
C00799=1047.622,-50.336,427.089,169.941,32.785,156.192
C00800=1047.615,-50.586,427.101,169.939,32.784,156.192
C00801=1047.608,-50.867,427.115,169.936,32.783,156.192
C00802=1047.601,-51.148,427.129,169.934,32.781,156.192
C00803=1047.594,-51.428,427.143,169.932,32.780,156.192
C00804=1047.586,-51.710,427.157,169.929,32.779,156.191
C00805=1047.580,-51.959,427.169,169.927,32.778,156.191
C00806=1047.574,-52.209,427.182,169.925,32.777,156.191
C00807=1047.567,-52.459,427.194,169.923,32.776,156.191
C00808=1047.561,-52.709,427.206,169.921,32.774,156.191
C00809=1047.554,-52.958,427.219,169.919,32.773,156.191
C00810=1047.548,-53.207,427.231,169.917,32.773,156.191
C00811=1047.542,-53.457,427.244,169.915,32.771,156.191
C00812=1047.535,-53.707,427.256,169.913,32.770,156.191
C00813=1047.529,-53.957,427.268,169.910,32.769,156.190
C00814=1047.523,-54.205,427.280,169.908,32.768,156.190
C00815=1047.516,-54.455,427.292,169.906,32.767,156.190
C00816=1047.511,-54.705,427.304,169.905,32.766,156.190
C00817=1047.504,-54.954,427.316,169.903,32.765,156.190
C00818=1047.498,-55.204,427.329,169.901,32.764,156.190
C00819=1047.491,-55.454,427.341,169.899,32.763,156.190
C00820=1047.485,-55.703,427.353,169.897,32.762,156.190
C00821=1047.479,-55.953,427.365,169.895,32.760,156.189
C00822=1047.472,-56.203,427.377,169.893,32.759,156.189
C00823=1047.466,-56.452,427.390,169.890,32.758,156.189
C00824=1047.459,-56.702,427.402,169.888,32.757,156.189
C00825=1047.453,-56.951,427.414,169.886,32.756,156.189
C00826=1047.447,-57.201,427.427,169.884,32.755,156.189
C00827=1047.440,-57.451,427.438,169.882,32.754,156.189
C00828=1047.434,-57.700,427.450,169.880,32.753,156.189
C00829=1047.428,-57.950,427.462,169.878,32.752,156.189
C00830=1047.422,-58.200,427.474,169.876,32.751,156.189
C00831=1047.416,-58.450,427.487,169.873,32.750,156.188
C00832=1047.409,-58.699,427.499,169.871,32.749,156.188
C00833=1047.403,-58.949,427.511,169.869,32.748,156.188
C00834=1047.397,-59.199,427.523,169.867,32.747,156.188
C00835=1047.391,-59.448,427.535,169.865,32.746,156.188
C00836=1047.384,-59.697,427.547,169.863,32.744,156.188
C00837=1047.378,-59.947,427.559,169.861,32.744,156.188
C00838=1047.371,-60.197,427.571,169.859,32.743,156.188
C00839=1047.365,-60.446,427.583,169.857,32.741,156.188
C00840=1047.359,-60.696,427.596,169.854,32.740,156.188
C00841=1047.353,-60.946,427.607,169.853,32.740,156.188
C00842=1047.346,-61.195,427.619,169.851,32.739,156.187
C00843=1047.341,-61.445,427.631,169.849,32.737,156.187
C00844=1047.334,-61.695,427.643,169.847,32.736,156.187
C00845=1047.327,-61.944,427.655,169.845,32.736,156.187
C00846=1047.322,-62.193,427.667,169.843,32.734,156.187
C00847=1047.316,-62.443,427.679,169.841,32.733,156.187
C00848=1047.309,-62.693,427.691,169.838,32.732,156.187
C00849=1047.303,-62.943,427.703,169.836,32.732,156.187
C00850=1047.296,-63.193,427.715,169.834,32.730,156.187
C00851=1047.290,-63.441,427.727,169.832,32.729,156.187
C00852=1047.285,-63.692,427.738,169.830,32.728,156.186
C00853=1047.278,-63.941,427.750,169.828,32.727,156.186
C00854=1047.271,-64.191,427.762,169.826,32.726,156.186
C00855=1047.266,-64.440,427.775,169.823,32.725,156.186
C00856=1047.260,-64.690,427.787,169.821,32.724,156.186
C00857=1047.253,-64.940,427.798,169.819,32.723,156.186
C00858=1047.247,-65.190,427.810,169.817,32.722,156.186
C00859=1047.241,-65.439,427.822,169.815,32.721,156.186
C00860=1047.235,-65.689,427.833,169.813,32.720,156.186
C00861=1047.228,-65.938,427.845,169.811,32.719,156.186
C00862=1047.223,-66.188,427.857,169.808,32.718,156.186
C00863=1047.216,-66.437,427.869,169.806,32.717,156.185
C00864=1047.210,-66.687,427.881,169.804,32.716,156.185
C00865=1047.203,-66.969,427.894,169.803,32.715,156.185
C00866=1047.196,-67.252,427.907,169.800,32.714,156.185
C00867=1047.189,-67.534,427.921,169.798,32.713,156.185
C00868=1047.182,-67.817,427.934,169.795,32.712,156.185
C00869=1047.176,-68.066,427.946,169.793,32.711,156.185
C00870=1047.170,-68.316,427.957,169.791,32.710,156.185
C00871=1047.164,-68.566,427.969,169.789,32.709,156.185
C00872=1047.158,-68.815,427.981,169.787,32.708,156.185
C00873=1047.152,-69.065,427.992,169.785,32.707,156.184
C00874=1047.145,-69.314,428.004,169.783,32.706,156.184
C00875=1047.140,-69.564,428.016,169.780,32.705,156.184
C00876=1047.133,-69.814,428.028,169.778,32.704,156.184
C00877=1047.127,-70.063,428.040,169.776,32.703,156.184
C00878=1047.122,-70.313,428.051,169.774,32.702,156.184
C00879=1047.115,-70.563,428.063,169.772,32.701,156.184
C00880=1047.109,-70.812,428.074,169.770,32.700,156.184
C00881=1047.103,-71.062,428.086,169.768,32.699,156.184
C00882=1047.097,-71.312,428.098,169.765,32.698,156.184
C00883=1047.091,-71.561,428.109,169.763,32.698,156.184
C00884=1047.085,-71.811,428.120,169.761,32.696,156.184
C00885=1047.079,-72.060,428.132,169.759,32.695,156.184
C00886=1047.072,-72.310,428.143,169.757,32.694,156.183
C00887=1047.066,-72.560,428.156,169.755,32.694,156.183
C00888=1047.061,-72.810,428.167,169.753,32.693,156.183
C00889=1047.054,-73.059,428.179,169.751,32.692,156.183
C00890=1047.048,-73.309,428.190,169.749,32.691,156.183
C00891=1047.042,-73.559,428.202,169.747,32.690,156.183
C00892=1047.037,-73.808,428.213,169.745,32.689,156.183
C00893=1047.030,-74.058,428.225,169.743,32.688,156.183
C00894=1047.024,-74.307,428.236,169.740,32.687,156.183
C00895=1047.018,-74.557,428.248,169.738,32.686,156.183
C00896=1047.011,-74.807,428.259,169.736,32.685,156.183
C00897=1047.006,-75.057,428.270,169.734,32.684,156.183
C00898=1046.999,-75.306,428.282,169.732,32.684,156.183
C00899=1046.993,-75.556,428.293,169.729,32.683,156.183
C00900=1046.987,-75.806,428.304,169.727,32.682,156.183
C00901=1046.981,-76.055,428.316,169.725,32.682,156.183
C00902=1046.974,-76.305,428.327,169.723,32.681,156.182
C00903=1046.968,-76.555,428.338,169.721,32.680,156.182
C00904=1046.962,-76.804,428.350,169.718,32.679,156.182
C00905=1046.956,-77.054,428.361,169.716,32.678,156.182
C00906=1046.950,-77.304,428.372,169.714,32.677,156.182
C00907=1046.943,-77.553,428.384,169.712,32.676,156.182
C00908=1046.938,-77.803,428.395,169.710,32.676,156.182
C00909=1046.931,-78.053,428.406,169.707,32.675,156.182
C00910=1046.925,-78.302,428.416,169.705,32.674,156.182
C00911=1046.918,-78.552,428.428,169.703,32.673,156.182
C00912=1046.912,-78.801,428.439,169.702,32.673,156.182
C00913=1046.906,-79.051,428.450,169.700,32.672,156.182
C00914=1046.900,-79.301,428.461,169.697,32.671,156.182
C00915=1046.894,-79.550,428.473,169.695,32.670,156.182
C00916=1046.888,-79.800,428.484,169.693,32.669,156.182
C00917=1046.882,-80.050,428.495,169.691,32.669,156.182
C00918=1046.876,-80.300,428.506,169.689,32.668,156.182
C00919=1046.869,-80.549,428.517,169.686,32.667,156.182
C00920=1046.863,-80.798,428.528,169.684,32.667,156.182
C00921=1046.856,-81.049,428.540,169.682,32.666,156.182
C00922=1046.851,-81.298,428.550,169.680,32.666,156.182
C00923=1046.844,-81.548,428.561,169.677,32.665,156.182
C00924=1046.838,-81.797,428.572,169.675,32.664,156.181
C00925=1046.831,-82.048,428.583,169.673,32.663,156.181
C00926=1046.825,-82.297,428.593,169.671,32.663,156.181
C00927=1046.819,-82.547,428.605,169.668,32.662,156.181
C00928=1046.813,-82.796,428.616,169.666,32.661,156.181
C00929=1046.805,-83.081,428.629,169.664,32.661,156.181
C00930=1046.798,-83.365,428.641,169.661,32.660,156.181
C00931=1046.792,-83.650,428.653,169.659,32.659,156.181
C00932=1046.784,-83.935,428.666,169.656,32.658,156.181
C00933=1046.777,-84.184,428.676,169.654,32.658,156.181
C00934=1046.771,-84.434,428.688,169.652,32.657,156.181
C00935=1046.765,-84.683,428.699,169.650,32.656,156.181
C00936=1046.759,-84.933,428.709,169.648,32.656,156.181
C00937=1046.752,-85.183,428.720,169.646,32.655,156.181
C00938=1046.747,-85.432,428.731,169.644,32.654,156.181
C00939=1046.740,-85.682,428.742,169.641,32.654,156.181
C00940=1046.734,-85.932,428.753,169.639,32.653,156.181
C00941=1046.728,-86.181,428.763,169.637,32.652,156.181
C00942=1046.722,-86.431,428.775,169.635,32.652,156.181
C00943=1046.715,-86.680,428.785,169.632,32.651,156.181
C00944=1046.709,-86.931,428.796,169.630,32.650,156.181
C00945=1046.703,-87.180,428.807,169.628,32.650,156.181
C00946=1046.697,-87.429,428.817,169.626,32.649,156.181
C00947=1046.690,-87.680,428.829,169.623,32.649,156.181
C00948=1046.685,-87.929,428.839,169.621,32.648,156.181
C00949=1046.678,-88.179,428.850,169.619,32.647,156.181
C00950=1046.672,-88.429,428.860,169.617,32.647,156.181
C00951=1046.666,-88.678,428.871,169.614,32.646,156.181
C00952=1046.659,-88.928,428.882,169.612,32.646,156.181
C00953=1046.654,-89.178,428.893,169.610,32.645,156.181
C00954=1046.647,-89.427,428.903,169.608,32.644,156.181
C00955=1046.641,-89.677,428.914,169.605,32.644,156.181
C00956=1046.635,-89.927,428.925,169.603,32.643,156.181
C00957=1046.629,-90.176,428.935,169.601,32.643,156.181
C00958=1046.623,-90.427,428.946,169.600,32.642,156.181
C00959=1046.617,-90.676,428.957,169.597,32.642,156.181
C00960=1046.610,-90.925,428.967,169.595,32.641,156.181
C00961=1046.605,-91.175,428.978,169.593,32.640,156.181
C00962=1046.598,-91.425,428.989,169.591,32.640,156.181
C00963=1046.592,-91.674,428.999,169.588,32.639,156.181
C00964=1046.586,-91.924,429.010,169.586,32.638,156.181
C00965=1046.579,-92.174,429.020,169.584,32.638,156.181
C00966=1046.574,-92.424,429.031,169.582,32.637,156.181
C00967=1046.568,-92.673,429.042,169.579,32.636,156.181
C00968=1046.562,-92.923,429.052,169.577,32.636,156.181
C00969=1046.555,-93.173,429.063,169.575,32.635,156.181
C00970=1046.549,-93.422,429.073,169.573,32.635,156.181
C00971=1046.543,-93.672,429.084,169.570,32.634,156.181
C00972=1046.538,-93.922,429.094,169.568,32.634,156.181
C00973=1046.531,-94.172,429.105,169.566,32.633,156.181
C00974=1046.525,-94.421,429.116,169.563,32.633,156.181
C00975=1046.518,-94.671,429.126,169.561,32.632,156.181
C00976=1046.513,-94.921,429.136,169.559,32.632,156.181
C00977=1046.507,-95.170,429.147,169.557,32.631,156.181
C00978=1046.500,-95.420,429.158,169.554,32.631,156.181
C00979=1046.495,-95.670,429.168,169.552,32.630,156.181
C00980=1046.488,-95.919,429.178,169.550,32.630,156.181
C00981=1046.482,-96.169,429.189,169.549,32.629,156.181
C00982=1046.477,-96.419,429.199,169.546,32.629,156.181
C00983=1046.470,-96.669,429.210,169.544,32.628,156.181
C00984=1046.464,-96.918,429.221,169.542,32.627,156.181
C00985=1046.458,-97.168,429.230,169.540,32.627,156.181
C00986=1046.452,-97.418,429.241,169.537,32.626,156.181
C00987=1046.446,-97.667,429.251,169.535,32.626,156.181
C00988=1046.440,-97.918,429.262,169.533,32.625,156.181
C00989=1046.434,-98.167,429.271,169.530,32.625,156.181
C00990=1046.427,-98.417,429.282,169.528,32.625,156.181
C00991=1046.421,-98.666,429.293,169.526,32.624,156.181
C00992=1046.415,-98.916,429.302,169.524,32.624,156.181
C00993=1046.408,-99.202,429.314,169.521,32.623,156.181
C00994=1046.401,-99.490,429.326,169.518,32.623,156.181
C00995=1046.394,-99.776,429.338,169.516,32.622,156.181
C00996=1046.386,-100.063,429.350,169.513,32.622,156.181
C00997=1046.380,-100.313,429.359,169.511,32.622,156.181
C00998=1046.375,-100.562,429.370,169.508,32.621,156.181
C00999=1046.368,-100.812,429.380,169.506,32.621,156.181
C01000=1046.361,-101.062,429.390,169.504,32.620,156.181
C01001=1046.356,-101.312,429.400,169.501,32.620,156.181
C01002=1046.350,-101.562,429.410,169.499,32.619,156.181
C01003=1046.343,-101.811,429.420,169.498,32.619,156.181
C01004=1046.338,-102.061,429.430,169.496,32.619,156.181
C01005=1046.331,-102.310,429.441,169.493,32.618,156.181
C01006=1046.325,-102.560,429.450,169.491,32.618,156.181
C01007=1046.319,-102.809,429.461,169.489,32.617,156.181
C01008=1046.313,-103.060,429.471,169.486,32.617,156.181
C01009=1046.306,-103.310,429.481,169.484,32.617,156.181
C01010=1046.301,-103.559,429.491,169.482,32.617,156.181
C01011=1046.295,-103.809,429.501,169.479,32.616,156.181
C01012=1046.288,-104.059,429.511,169.477,32.615,156.181
C01013=1046.282,-104.308,429.521,169.475,32.615,156.181
C01014=1046.276,-104.558,429.531,169.473,32.615,156.181
C01015=1046.270,-104.807,429.541,169.470,32.615,156.181
C01016=1046.264,-105.057,429.551,169.468,32.615,156.182
C01017=1046.258,-105.307,429.561,169.466,32.614,156.182
C01018=1046.252,-105.557,429.571,169.463,32.614,156.182
C01019=1046.246,-105.806,429.581,169.461,32.613,156.182
C01020=1046.240,-106.056,429.590,169.459,32.613,156.182
C01021=1046.234,-106.306,429.601,169.456,32.613,156.182
C01022=1046.228,-106.555,429.611,169.454,32.612,156.182
C01023=1046.221,-106.806,429.621,169.452,32.612,156.182
C01024=1046.215,-107.056,429.630,169.449,32.612,156.182
C01025=1046.208,-107.305,429.640,169.447,32.612,156.182
C01026=1046.203,-107.555,429.651,169.445,32.611,156.182
C01027=1046.197,-107.805,429.660,169.443,32.611,156.182
C01028=1046.190,-108.054,429.670,169.441,32.611,156.182
C01029=1046.184,-108.304,429.680,169.439,32.611,156.182
C01030=1046.178,-108.553,429.690,169.436,32.610,156.182
C01031=1046.172,-108.803,429.699,169.434,32.610,156.182
C01032=1046.165,-109.053,429.709,169.432,32.610,156.182
C01033=1046.159,-109.303,429.719,169.429,32.610,156.182
C01034=1046.154,-109.553,429.729,169.427,32.609,156.182
C01035=1046.148,-109.803,429.738,169.425,32.609,156.182
C01036=1046.141,-110.052,429.749,169.423,32.609,156.183
C01037=1046.135,-110.302,429.758,169.420,32.609,156.183
C01038=1046.129,-110.551,429.768,169.418,32.609,156.183
C01039=1046.123,-110.801,429.777,169.416,32.608,156.183
C01040=1046.116,-111.051,429.787,169.413,32.608,156.183
C01041=1046.110,-111.301,429.796,169.411,32.608,156.183
C01042=1046.104,-111.551,429.806,169.409,32.608,156.183
C01043=1046.098,-111.800,429.816,169.406,32.607,156.183
C01044=1046.092,-112.050,429.825,169.404,32.607,156.183
C01045=1046.086,-112.299,429.835,169.402,32.607,156.183
C01046=1046.080,-112.549,429.845,169.399,32.607,156.183
C01047=1046.074,-112.799,429.855,169.397,32.607,156.183
C01048=1046.068,-113.048,429.864,169.395,32.607,156.183
C01049=1046.062,-113.298,429.874,169.392,32.606,156.183
C01050=1046.056,-113.548,429.883,169.391,32.606,156.183
C01051=1046.050,-113.798,429.893,169.389,32.606,156.183
C01052=1046.043,-114.048,429.903,169.386,32.606,156.183
C01053=1046.037,-114.297,429.912,169.384,32.606,156.184
C01054=1046.031,-114.547,429.922,169.381,32.605,156.184
C01055=1046.025,-114.797,429.931,169.379,32.605,156.184
C01056=1046.019,-115.047,429.941,169.377,32.605,156.184
C01057=1046.012,-115.332,429.951,169.374,32.605,156.184
C01058=1046.005,-115.618,429.962,169.371,32.605,156.184
C01059=1045.998,-115.903,429.973,169.369,32.605,156.184
C01060=1045.991,-116.190,429.984,169.366,32.605,156.184
C01061=1045.985,-116.440,429.993,169.364,32.605,156.184
C01062=1045.979,-116.690,430.003,169.361,32.604,156.184
C01063=1045.973,-116.939,430.012,169.359,32.604,156.184
C01064=1045.967,-117.188,430.022,169.357,32.604,156.184
C01065=1045.961,-117.438,430.031,169.354,32.604,156.185
C01066=1045.954,-117.688,430.040,169.352,32.604,156.185
C01067=1045.948,-117.938,430.050,169.350,32.604,156.185
C01068=1045.942,-118.187,430.059,169.347,32.604,156.185
C01069=1045.936,-118.438,430.068,169.345,32.604,156.185
C01070=1045.930,-118.687,430.077,169.343,32.604,156.185
C01071=1045.924,-118.937,430.087,169.340,32.603,156.185
C01072=1045.918,-119.186,430.097,169.338,32.604,156.185
C01073=1045.912,-119.436,430.106,169.336,32.604,156.185
C01074=1045.905,-119.686,430.116,169.334,32.603,156.185
C01075=1045.899,-119.936,430.124,169.332,32.604,156.185
C01076=1045.893,-120.185,430.133,169.329,32.603,156.186
C01077=1045.887,-120.435,430.143,169.327,32.603,156.186
C01078=1045.881,-120.685,430.152,169.325,32.604,156.186
C01079=1045.875,-120.935,430.162,169.322,32.603,156.186
C01080=1045.869,-121.185,430.171,169.320,32.603,156.186
C01081=1045.863,-121.434,430.180,169.318,32.604,156.186
C01082=1045.856,-121.684,430.189,169.315,32.603,156.186
C01083=1045.850,-121.933,430.198,169.313,32.603,156.186
C01084=1045.844,-122.184,430.207,169.310,32.603,156.186
C01085=1045.838,-122.434,430.217,169.308,32.603,156.186
C01086=1045.833,-122.683,430.226,169.306,32.604,156.186
C01087=1045.827,-122.933,430.235,169.303,32.603,156.187
C01088=1045.820,-123.183,430.244,169.301,32.603,156.187
C01089=1045.814,-123.432,430.253,169.299,32.603,156.187
C01090=1045.808,-123.682,430.263,169.296,32.603,156.187
C01091=1045.802,-123.932,430.272,169.294,32.604,156.187
C01092=1045.796,-124.182,430.281,169.292,32.603,156.187
C01093=1045.789,-124.431,430.290,169.289,32.603,156.187
C01094=1045.784,-124.681,430.299,169.287,32.603,156.187
C01095=1045.778,-124.931,430.308,169.284,32.603,156.187
C01096=1045.772,-125.181,430.317,169.282,32.604,156.187
C01097=1045.765,-125.431,430.326,169.280,32.603,156.188
C01098=1045.759,-125.680,430.335,169.278,32.604,156.188
C01099=1045.753,-125.930,430.344,169.276,32.604,156.188
C01100=1045.747,-126.180,430.353,169.274,32.604,156.188
C01101=1045.741,-126.430,430.362,169.271,32.604,156.188
C01102=1045.735,-126.679,430.371,169.269,32.604,156.188
C01103=1045.728,-126.929,430.380,169.266,32.604,156.188
C01104=1045.722,-127.179,430.389,169.264,32.604,156.188
C01105=1045.717,-127.428,430.398,169.262,32.605,156.189
C01106=1045.710,-127.678,430.406,169.259,32.604,156.189
C01107=1045.705,-127.927,430.416,169.257,32.605,156.189
C01108=1045.699,-128.177,430.426,169.255,32.604,156.189
C01109=1045.696,-128.428,430.437,169.253,32.603,156.189
C01110=1045.693,-128.677,430.447,169.251,32.602,156.188
C01111=1045.690,-128.927,430.459,169.249,32.599,156.188
C01112=1045.689,-129.177,430.471,169.247,32.597,156.188
C01113=1045.689,-129.428,430.484,169.245,32.595,156.188
C01114=1045.690,-129.679,430.497,169.244,32.591,156.187
C01115=1045.692,-129.928,430.511,169.242,32.587,156.186
C01116=1045.695,-130.178,430.526,169.241,32.583,156.186
C01117=1045.699,-130.429,430.541,169.240,32.579,156.185
C01118=1045.703,-130.680,430.557,169.240,32.574,156.184
C01119=1045.708,-130.930,430.574,169.239,32.568,156.183
C01120=1045.714,-131.179,430.591,169.238,32.562,156.182
C01121=1045.358,-131.203,430.350,169.192,32.741,156.215
C01122=1045.352,-130.953,430.333,169.192,32.747,156.216
C01123=1045.346,-130.703,430.317,169.193,32.752,156.217
C01124=1045.342,-130.453,430.301,169.194,32.757,156.217
C01125=1045.338,-130.202,430.286,169.196,32.762,156.218
C01126=1045.335,-129.952,430.271,169.197,32.767,156.219
C01127=1045.333,-129.702,430.256,169.198,32.770,156.219
C01128=1045.333,-129.451,430.243,169.200,32.773,156.220
C01129=1045.333,-129.201,430.230,169.201,32.777,156.220
C01130=1045.334,-128.951,430.218,169.202,32.779,156.221
C01131=1045.336,-128.701,430.206,169.204,32.781,156.221
C01132=1045.339,-128.451,430.195,169.206,32.782,156.221
C01133=1045.343,-128.202,430.185,169.208,32.783,156.221
C01134=1045.348,-127.951,430.176,169.210,32.783,156.221
C01135=1045.354,-127.702,430.166,169.213,32.784,156.221
C01136=1045.359,-127.453,430.157,169.215,32.783,156.221
C01137=1045.365,-127.202,430.148,169.218,32.784,156.221
C01138=1045.372,-126.953,430.139,169.220,32.783,156.221
C01139=1045.377,-126.703,430.130,169.222,32.783,156.221
C01140=1045.384,-126.453,430.121,169.225,32.783,156.221
C01141=1045.391,-126.204,430.112,169.227,32.783,156.220
C01142=1045.396,-125.954,430.103,169.229,32.783,156.220
C01143=1045.402,-125.704,430.094,169.232,32.783,156.220
C01144=1045.409,-125.454,430.086,169.234,32.783,156.220
C01145=1045.415,-125.204,430.076,169.237,32.782,156.220
C01146=1045.420,-124.955,430.067,169.239,32.782,156.220
C01147=1045.426,-124.705,430.058,169.241,32.782,156.220
C01148=1045.433,-124.455,430.049,169.244,32.782,156.220
C01149=1045.439,-124.205,430.039,169.246,32.782,156.219
C01150=1045.445,-123.956,430.031,169.249,32.782,156.219
C01151=1045.451,-123.706,430.021,169.251,32.782,156.219
C01152=1045.458,-123.456,430.012,169.253,32.782,156.219
C01153=1045.463,-123.206,430.004,169.256,32.782,156.219
C01154=1045.469,-122.957,429.994,169.258,32.782,156.219
C01155=1045.475,-122.707,429.985,169.259,32.782,156.219
C01156=1045.481,-122.457,429.976,169.262,32.782,156.219
C01157=1045.487,-122.207,429.966,169.264,32.782,156.219
C01158=1045.494,-121.958,429.958,169.267,32.782,156.219
C01159=1045.500,-121.708,429.948,169.269,32.782,156.219
C01160=1045.506,-121.458,429.939,169.271,32.782,156.218
C01161=1045.512,-121.208,429.930,169.274,32.782,156.218
C01162=1045.518,-120.958,429.920,169.276,32.782,156.218
C01163=1045.524,-120.709,429.911,169.278,32.782,156.218
C01164=1045.530,-120.459,429.903,169.281,32.782,156.218
C01165=1045.536,-120.209,429.893,169.283,32.782,156.218
C01166=1045.542,-119.960,429.884,169.286,32.782,156.218
C01167=1045.549,-119.710,429.874,169.288,32.782,156.218
C01168=1045.554,-119.461,429.865,169.290,32.782,156.218
C01169=1045.560,-119.210,429.856,169.293,32.782,156.218
C01170=1045.566,-118.960,429.846,169.295,32.782,156.217
C01171=1045.572,-118.711,429.837,169.297,32.782,156.217
C01172=1045.579,-118.461,429.827,169.300,32.782,156.217
C01173=1045.585,-118.211,429.818,169.302,32.782,156.217
C01174=1045.591,-117.962,429.809,169.304,32.782,156.217
C01175=1045.597,-117.712,429.800,169.307,32.782,156.217
C01176=1045.603,-117.462,429.791,169.309,32.782,156.217
C01177=1045.609,-117.212,429.781,169.312,32.782,156.217
C01178=1045.615,-116.962,429.772,169.314,32.782,156.217
C01179=1045.622,-116.713,429.762,169.316,32.783,156.217
C01180=1045.628,-116.463,429.752,169.318,32.782,156.217
C01181=1045.633,-116.214,429.743,169.320,32.782,156.217
C01182=1045.641,-115.927,429.733,169.323,32.783,156.217
C01183=1045.648,-115.641,429.721,169.325,32.783,156.216
C01184=1045.655,-115.357,429.711,169.328,32.783,156.216
C01185=1045.662,-115.070,429.700,169.331,32.783,156.216
C01186=1045.668,-114.820,429.690,169.333,32.783,156.216
C01187=1045.674,-114.570,429.681,169.336,32.783,156.216
C01188=1045.680,-114.321,429.671,169.338,32.783,156.216
C01189=1045.686,-114.071,429.662,169.340,32.783,156.216
C01190=1045.692,-113.822,429.652,169.343,32.784,156.216
C01191=1045.698,-113.572,429.643,169.345,32.784,156.216
C01192=1045.704,-113.322,429.633,169.347,32.784,156.216
C01193=1045.710,-113.072,429.624,169.350,32.784,156.216
C01194=1045.717,-112.822,429.614,169.352,32.784,156.216
C01195=1045.723,-112.573,429.605,169.354,32.784,156.215
C01196=1045.729,-112.323,429.595,169.357,32.784,156.215
C01197=1045.735,-112.074,429.585,169.359,32.784,156.215
C01198=1045.742,-111.824,429.575,169.361,32.785,156.215
C01199=1045.748,-111.574,429.566,169.364,32.785,156.215
C01200=1045.753,-111.324,429.555,169.366,32.785,156.215
C01201=1045.759,-111.074,429.546,169.368,32.785,156.215
C01202=1045.766,-110.824,429.536,169.371,32.786,156.215
C01203=1045.772,-110.575,429.527,169.373,32.786,156.215
C01204=1045.778,-110.325,429.517,169.375,32.786,156.215
C01205=1045.784,-110.075,429.508,169.377,32.786,156.215
C01206=1045.791,-109.826,429.497,169.379,32.787,156.215
C01207=1045.797,-109.576,429.488,169.381,32.786,156.215
C01208=1045.803,-109.326,429.478,169.384,32.786,156.215
C01209=1045.809,-109.076,429.469,169.386,32.787,156.215
C01210=1045.815,-108.827,429.459,169.388,32.787,156.215
C01211=1045.821,-108.576,429.449,169.391,32.787,156.215
C01212=1045.827,-108.327,429.439,169.393,32.787,156.214
C01213=1045.833,-108.078,429.429,169.395,32.788,156.214
C01214=1045.840,-107.828,429.419,169.398,32.788,156.214
C01215=1045.846,-107.578,429.410,169.400,32.788,156.214
C01216=1045.852,-107.328,429.400,169.402,32.788,156.214
C01217=1045.858,-107.079,429.390,169.405,32.789,156.214
C01218=1045.864,-106.829,429.380,169.407,32.789,156.214
C01219=1045.870,-106.579,429.370,169.409,32.789,156.214
C01220=1045.876,-106.330,429.360,169.412,32.789,156.214
C01221=1045.883,-106.080,429.350,169.414,32.790,156.214
C01222=1045.888,-105.830,429.340,169.416,32.790,156.214
C01223=1045.894,-105.580,429.331,169.419,32.791,156.214
C01224=1045.901,-105.331,429.320,169.421,32.791,156.214
C01225=1045.907,-105.081,429.311,169.423,32.791,156.214
C01226=1045.912,-104.831,429.301,169.426,32.791,156.214
C01227=1045.919,-104.582,429.290,169.428,32.791,156.214
C01228=1045.925,-104.332,429.281,169.430,32.792,156.214
C01229=1045.931,-104.082,429.271,169.432,32.792,156.214
C01230=1045.937,-103.832,429.260,169.434,32.793,156.214
C01231=1045.944,-103.582,429.251,169.436,32.793,156.214
C01232=1045.950,-103.333,429.240,169.439,32.793,156.214
C01233=1045.956,-103.083,429.230,169.441,32.794,156.214
C01234=1045.962,-102.833,429.221,169.443,32.794,156.214
C01235=1045.968,-102.584,429.210,169.446,32.794,156.214
C01236=1045.974,-102.334,429.200,169.448,32.795,156.214
C01237=1045.980,-102.085,429.190,169.450,32.795,156.214
C01238=1045.986,-101.835,429.180,169.452,32.795,156.213
C01239=1045.992,-101.585,429.171,169.455,32.796,156.213
C01240=1045.999,-101.335,429.159,169.457,32.796,156.213
C01241=1046.005,-101.085,429.150,169.459,32.797,156.213
C01242=1046.011,-100.836,429.140,169.462,32.797,156.213
C01243=1046.017,-100.586,429.129,169.464,32.797,156.213
C01244=1046.023,-100.337,429.119,169.466,32.797,156.213
C01245=1046.029,-100.087,429.110,169.469,32.798,156.213
C01246=1046.036,-99.800,429.097,169.471,32.798,156.213
C01247=1046.044,-99.513,429.086,169.474,32.799,156.213
C01248=1046.051,-99.227,429.074,169.477,32.799,156.213
C01249=1046.058,-98.940,429.062,169.479,32.799,156.213
C01250=1046.064,-98.690,429.052,169.482,32.800,156.213
C01251=1046.070,-98.441,429.042,169.484,32.800,156.213
C01252=1046.076,-98.190,429.031,169.486,32.801,156.213
C01253=1046.083,-97.941,429.021,169.488,32.801,156.213
C01254=1046.089,-97.691,429.011,169.490,32.802,156.213
C01255=1046.095,-97.441,429.001,169.492,32.802,156.213
C01256=1046.101,-97.192,428.990,169.494,32.802,156.213
C01257=1046.107,-96.941,428.980,169.497,32.803,156.213
C01258=1046.114,-96.692,428.969,169.499,32.803,156.213
C01259=1046.119,-96.442,428.959,169.501,32.804,156.213
C01260=1046.125,-96.193,428.948,169.503,32.804,156.213
C01261=1046.131,-95.943,428.938,169.506,32.805,156.213
C01262=1046.137,-95.693,428.928,169.508,32.805,156.213
C01263=1046.144,-95.443,428.917,169.510,32.806,156.213
C01264=1046.150,-95.194,428.906,169.513,32.807,156.213
C01265=1046.155,-94.944,428.896,169.515,32.807,156.213
C01266=1046.161,-94.695,428.886,169.517,32.808,156.213
C01267=1046.168,-94.444,428.875,169.519,32.808,156.213
C01268=1046.174,-94.195,428.864,169.522,32.809,156.213
C01269=1046.180,-93.945,428.854,169.524,32.809,156.213
C01270=1046.185,-93.696,428.843,169.526,32.810,156.213
C01271=1046.193,-93.446,428.833,169.528,32.810,156.213
C01272=1046.198,-93.196,428.823,169.531,32.811,156.213
C01273=1046.204,-92.946,428.812,169.533,32.811,156.213
C01274=1046.210,-92.697,428.801,169.535,32.812,156.213
C01275=1046.217,-92.447,428.790,169.538,32.812,156.213
C01276=1046.223,-92.197,428.781,169.540,32.813,156.213
C01277=1046.228,-91.948,428.770,169.542,32.813,156.213
C01278=1046.235,-91.698,428.759,169.544,32.814,156.213
C01279=1046.241,-91.448,428.748,169.546,32.814,156.213
C01280=1046.247,-91.199,428.737,169.548,32.815,156.213
C01281=1046.253,-90.949,428.727,169.550,32.815,156.213
C01282=1046.259,-90.699,428.717,169.552,32.816,156.213
C01283=1046.265,-90.449,428.706,169.555,32.816,156.213
C01284=1046.272,-90.200,428.695,169.557,32.817,156.213
C01285=1046.277,-89.951,428.684,169.559,32.818,156.213
C01286=1046.284,-89.700,428.673,169.561,32.818,156.213
C01287=1046.290,-89.451,428.663,169.564,32.819,156.213
C01288=1046.296,-89.201,428.653,169.566,32.819,156.213
C01289=1046.303,-88.951,428.642,169.568,32.820,156.213
C01290=1046.309,-88.702,428.631,169.570,32.821,156.213
C01291=1046.314,-88.452,428.620,169.573,32.821,156.213
C01292=1046.321,-88.202,428.610,169.575,32.822,156.213
C01293=1046.327,-87.953,428.599,169.577,32.822,156.213
C01294=1046.333,-87.703,428.588,169.580,32.823,156.213
C01295=1046.340,-87.453,428.577,169.582,32.824,156.213
C01296=1046.346,-87.204,428.566,169.584,32.824,156.213
C01297=1046.352,-86.954,428.555,169.586,32.825,156.213
C01298=1046.358,-86.705,428.545,169.589,32.826,156.213
C01299=1046.364,-86.455,428.534,169.591,32.826,156.213
C01300=1046.371,-86.205,428.523,169.593,32.827,156.213
C01301=1046.377,-85.956,428.513,169.595,32.827,156.213
C01302=1046.383,-85.706,428.501,169.598,32.828,156.213
C01303=1046.389,-85.456,428.490,169.600,32.829,156.213
C01304=1046.396,-85.207,428.480,169.601,32.829,156.213
C01305=1046.402,-84.957,428.469,169.603,32.830,156.213
C01306=1046.408,-84.707,428.458,169.606,32.831,156.213
C01307=1046.414,-84.457,428.447,169.608,32.831,156.213
C01308=1046.420,-84.208,428.436,169.610,32.832,156.213
C01309=1046.427,-83.958,428.425,169.612,32.832,156.214
C01310=1046.434,-83.673,428.413,169.615,32.833,156.213
C01311=1046.441,-83.389,428.401,169.617,32.834,156.214
C01312=1046.448,-83.104,428.388,169.620,32.834,156.214
C01313=1046.455,-82.820,428.376,169.623,32.835,156.214
C01314=1046.462,-82.570,428.365,169.625,32.836,156.214
C01315=1046.468,-82.320,428.354,169.627,32.836,156.214
C01316=1046.474,-82.070,428.343,169.629,32.837,156.214
C01317=1046.480,-81.821,428.332,169.632,32.838,156.214
C01318=1046.486,-81.571,428.322,169.634,32.838,156.214
C01319=1046.493,-81.322,428.310,169.636,32.839,156.214
C01320=1046.499,-81.072,428.299,169.638,32.839,156.214
C01321=1046.505,-80.822,428.288,169.640,32.840,156.214
C01322=1046.512,-80.572,428.277,169.643,32.841,156.214
C01323=1046.518,-80.323,428.266,169.645,32.841,156.214
C01324=1046.524,-80.073,428.255,169.647,32.842,156.214
C01325=1046.531,-79.824,428.244,169.649,32.843,156.214
C01326=1046.537,-79.574,428.233,169.652,32.844,156.214
C01327=1046.543,-79.324,428.222,169.654,32.844,156.214
C01328=1046.549,-79.074,428.211,169.656,32.845,156.214
C01329=1046.555,-78.825,428.200,169.657,32.846,156.214
C01330=1046.562,-78.575,428.188,169.659,32.847,156.214
C01331=1046.568,-78.326,428.177,169.662,32.848,156.214
C01332=1046.574,-78.075,428.166,169.664,32.848,156.214
C01333=1046.580,-77.827,428.154,169.666,32.849,156.214
C01334=1046.586,-77.576,428.143,169.668,32.849,156.214
C01335=1046.592,-77.327,428.132,169.671,32.850,156.214
C01336=1046.598,-77.077,428.121,169.673,32.851,156.214
C01337=1046.604,-76.828,428.109,169.675,32.852,156.214
C01338=1046.611,-76.578,428.098,169.677,32.853,156.215
C01339=1046.616,-76.328,428.087,169.679,32.854,156.215
C01340=1046.623,-76.079,428.075,169.682,32.855,156.215
C01341=1046.629,-75.828,428.064,169.684,32.855,156.215
C01342=1046.635,-75.579,428.053,169.686,32.856,156.215
C01343=1046.642,-75.329,428.041,169.688,32.857,156.215
C01344=1046.648,-75.080,428.030,169.690,32.857,156.215
C01345=1046.654,-74.830,428.019,169.693,32.858,156.215
C01346=1046.660,-74.581,428.007,169.695,32.859,156.215
C01347=1046.666,-74.331,427.996,169.697,32.860,156.215
C01348=1046.673,-74.081,427.984,169.699,32.861,156.215
C01349=1046.679,-73.831,427.973,169.701,32.861,156.215
C01350=1046.685,-73.582,427.961,169.704,32.862,156.215
C01351=1046.691,-73.332,427.950,169.706,32.863,156.215
C01352=1046.697,-73.082,427.939,169.708,32.864,156.215
C01353=1046.703,-72.833,427.927,169.710,32.865,156.215
C01354=1046.709,-72.583,427.916,169.712,32.866,156.216
C01355=1046.716,-72.333,427.904,169.714,32.867,156.216
C01356=1046.721,-72.084,427.893,169.716,32.868,156.216
C01357=1046.727,-71.834,427.880,169.718,32.869,156.216
C01358=1046.733,-71.584,427.869,169.720,32.870,156.216
C01359=1046.740,-71.335,427.857,169.722,32.871,156.216
C01360=1046.746,-71.086,427.846,169.724,32.871,156.216
C01361=1046.751,-70.835,427.834,169.726,32.872,156.216
C01362=1046.758,-70.586,427.822,169.729,32.874,156.216
C01363=1046.764,-70.336,427.811,169.731,32.875,156.216
C01364=1046.770,-70.087,427.799,169.733,32.875,156.216
C01365=1046.776,-69.836,427.787,169.735,32.876,156.216
C01366=1046.782,-69.587,427.776,169.737,32.877,156.216
C01367=1046.788,-69.337,427.764,169.739,32.878,156.217
C01368=1046.794,-69.088,427.753,169.741,32.879,156.217
C01369=1046.800,-68.838,427.740,169.744,32.880,156.217
C01370=1046.807,-68.588,427.729,169.746,32.881,156.217
C01371=1046.813,-68.339,427.717,169.748,32.882,156.217
C01372=1046.819,-68.090,427.706,169.750,32.883,156.217
C01373=1046.825,-67.839,427.694,169.752,32.884,156.217
C01374=1046.832,-67.557,427.680,169.755,32.885,156.217
C01375=1046.839,-67.275,427.667,169.757,32.886,156.217
C01376=1046.847,-66.993,427.654,169.760,32.887,156.217
C01377=1046.853,-66.710,427.641,169.762,32.888,156.217
C01378=1046.859,-66.461,427.629,169.764,32.889,156.218
C01379=1046.865,-66.211,427.617,169.766,32.890,156.218
C01380=1046.872,-65.961,427.605,169.768,32.891,156.218
C01381=1046.878,-65.711,427.593,169.771,32.892,156.218
C01382=1046.884,-65.463,427.581,169.773,32.893,156.218
C01383=1046.890,-65.212,427.570,169.774,32.894,156.218
C01384=1046.897,-64.963,427.558,169.776,32.895,156.218
C01385=1046.902,-64.714,427.546,169.778,32.896,156.218
C01386=1046.908,-64.464,427.534,169.780,32.896,156.218
C01387=1046.915,-64.214,427.523,169.782,32.898,156.218
C01388=1046.921,-63.964,427.510,169.785,32.899,156.218
C01389=1046.927,-63.715,427.499,169.787,32.900,156.218
C01390=1046.933,-63.465,427.487,169.789,32.900,156.219
C01391=1046.939,-63.215,427.475,169.791,32.902,156.219
C01392=1046.946,-62.965,427.463,169.793,32.903,156.219
C01393=1046.952,-62.717,427.451,169.795,32.904,156.219
C01394=1046.958,-62.467,427.439,169.797,32.904,156.219
C01395=1046.964,-62.217,427.427,169.800,32.906,156.219
C01396=1046.971,-61.968,427.415,169.802,32.907,156.219
C01397=1046.977,-61.717,427.403,169.804,32.908,156.219
C01398=1046.983,-61.468,427.391,169.806,32.908,156.219
C01399=1046.989,-61.219,427.379,169.808,32.910,156.219
C01400=1046.995,-60.969,427.367,169.810,32.911,156.220
C01401=1047.002,-60.719,427.355,169.812,32.912,156.220
C01402=1047.008,-60.470,427.343,169.815,32.912,156.220
C01403=1047.014,-60.220,427.330,169.817,32.914,156.220
C01404=1047.020,-59.970,427.319,169.819,32.915,156.220
C01405=1047.027,-59.721,427.308,169.821,32.916,156.220
C01406=1047.033,-59.471,427.295,169.823,32.916,156.220
C01407=1047.039,-59.221,427.283,169.825,32.918,156.220
C01408=1047.046,-58.972,427.271,169.827,32.919,156.220
C01409=1047.052,-58.722,427.258,169.829,32.919,156.220
C01410=1047.058,-58.473,427.247,169.832,32.921,156.221
C01411=1047.065,-58.223,427.235,169.834,32.922,156.221
C01412=1047.070,-57.973,427.222,169.835,32.923,156.221
C01413=1047.077,-57.724,427.210,169.837,32.923,156.221
C01414=1047.083,-57.474,427.198,169.839,32.925,156.221
C01415=1047.090,-57.224,427.186,169.841,32.926,156.221
C01416=1047.096,-56.975,427.174,169.843,32.927,156.221
C01417=1047.102,-56.725,427.161,169.845,32.928,156.221
C01418=1047.109,-56.475,427.149,169.848,32.929,156.221
C01419=1047.115,-56.226,427.137,169.850,32.930,156.221
C01420=1047.121,-55.977,427.125,169.852,32.931,156.222
C01421=1047.127,-55.727,427.113,169.854,32.932,156.222
C01422=1047.133,-55.477,427.101,169.856,32.933,156.222
C01423=1047.140,-55.228,427.089,169.858,32.934,156.222
C01424=1047.147,-54.978,427.077,169.860,32.935,156.222
C01425=1047.153,-54.728,427.064,169.862,32.936,156.222
C01426=1047.159,-54.478,427.052,169.864,32.937,156.222
C01427=1047.165,-54.229,427.040,169.867,32.938,156.222
C01428=1047.172,-53.979,427.028,169.869,32.939,156.222
C01429=1047.179,-53.730,427.015,169.871,32.941,156.222
C01430=1047.185,-53.480,427.003,169.873,32.941,156.223
C01431=1047.191,-53.231,426.991,169.875,32.942,156.223
C01432=1047.197,-52.981,426.978,169.877,32.944,156.223
C01433=1047.204,-52.731,426.966,169.879,32.944,156.223
C01434=1047.210,-52.482,426.954,169.881,32.945,156.223
C01435=1047.216,-52.232,426.942,169.883,32.947,156.223
C01436=1047.223,-51.982,426.930,169.885,32.948,156.223
C01437=1047.229,-51.733,426.916,169.888,32.948,156.223
C01438=1047.236,-51.452,426.904,169.890,32.950,156.223
C01439=1047.244,-51.170,426.889,169.892,32.951,156.224
C01440=1047.251,-50.890,426.875,169.895,32.952,156.224
C01441=1047.259,-50.609,426.861,169.896,32.954,156.224
C01442=1047.265,-50.359,426.849,169.898,32.955,156.224
C01443=1047.270,-50.109,426.836,169.900,32.956,156.224
C01444=1047.277,-49.860,426.824,169.902,32.957,156.224
C01445=1047.283,-49.610,426.811,169.904,32.958,156.224
C01446=1047.289,-49.360,426.798,169.906,32.959,156.224
C01447=1047.295,-49.110,426.786,169.908,32.961,156.225
C01448=1047.302,-48.861,426.773,169.910,32.962,156.225
C01449=1047.308,-48.611,426.761,169.913,32.963,156.225
C01450=1047.314,-48.362,426.748,169.915,32.964,156.225
C01451=1047.320,-48.112,426.735,169.917,32.966,156.225
C01452=1047.327,-47.863,426.723,169.919,32.967,156.225
C01453=1047.333,-47.613,426.710,169.921,32.968,156.225
C01454=1047.339,-47.364,426.697,169.923,32.969,156.226
C01455=1047.345,-47.114,426.684,169.925,32.970,156.226
C01456=1047.351,-46.864,426.673,169.927,32.972,156.226
C01457=1047.358,-46.615,426.659,169.929,32.973,156.226
C01458=1047.364,-46.365,426.647,169.931,32.974,156.226
C01459=1047.370,-46.116,426.633,169.933,32.975,156.226
C01460=1047.376,-45.866,426.621,169.935,32.976,156.226
C01461=1047.382,-45.616,426.609,169.937,32.978,156.227
C01462=1047.389,-45.367,426.596,169.939,32.979,156.227
C01463=1047.394,-45.117,426.583,169.941,32.980,156.227
C01464=1047.401,-44.868,426.570,169.943,32.981,156.227
C01465=1047.407,-44.618,426.558,169.945,32.982,156.227
C01466=1047.413,-44.368,426.545,169.947,32.984,156.227
C01467=1047.419,-44.119,426.532,169.949,32.985,156.227
C01468=1047.425,-43.869,426.519,169.951,32.986,156.228
C01469=1047.432,-43.619,426.506,169.954,32.987,156.228
C01470=1047.439,-43.370,426.494,169.956,32.989,156.228
C01471=1047.445,-43.120,426.481,169.958,32.990,156.228
C01472=1047.451,-42.871,426.468,169.960,32.991,156.228
C01473=1047.457,-42.621,426.455,169.962,32.993,156.228
C01474=1047.463,-42.371,426.442,169.964,32.993,156.228
C01475=1047.470,-42.122,426.430,169.965,32.995,156.229
C01476=1047.476,-41.873,426.417,169.967,32.996,156.229
C01477=1047.483,-41.623,426.403,169.969,32.997,156.229
C01478=1047.489,-41.373,426.391,169.971,32.999,156.229
C01479=1047.495,-41.123,426.378,169.973,33.000,156.229
C01480=1047.501,-40.874,426.364,169.975,33.001,156.229
C01481=1047.508,-40.625,426.352,169.977,33.002,156.229
C01482=1047.514,-40.375,426.339,169.979,33.004,156.230
C01483=1047.520,-40.125,426.327,169.981,33.005,156.230
C01484=1047.527,-39.875,426.313,169.983,33.006,156.230
C01485=1047.533,-39.626,426.300,169.985,33.007,156.230
C01486=1047.539,-39.376,426.287,169.987,33.008,156.230
C01487=1047.546,-39.127,426.274,169.989,33.010,156.230
C01488=1047.552,-38.878,426.262,169.991,33.011,156.230
C01489=1047.558,-38.628,426.248,169.993,33.013,156.231
C01490=1047.565,-38.378,426.235,169.995,33.013,156.231
C01491=1047.571,-38.128,426.222,169.997,33.015,156.231
C01492=1047.577,-37.879,426.209,169.999,33.016,156.231
C01493=1047.583,-37.630,426.196,170.001,33.018,156.231
C01494=1047.589,-37.380,426.183,170.003,33.019,156.231
C01495=1047.595,-37.131,426.170,170.005,33.021,156.232
C01496=1047.602,-36.881,426.156,170.007,33.021,156.232
C01497=1047.608,-36.632,426.143,170.009,33.023,156.232
C01498=1047.613,-36.381,426.130,170.011,33.024,156.232
C01499=1047.620,-36.132,426.117,170.013,33.026,156.232
C01500=1047.626,-35.883,426.103,170.015,33.027,156.232
C01501=1047.633,-35.633,426.090,170.017,33.029,156.233
C01502=1047.639,-35.352,426.076,170.019,33.030,156.233
C01503=1047.646,-35.072,426.061,170.022,33.032,156.233
C01504=1047.653,-34.791,426.045,170.024,33.033,156.233
C01505=1047.660,-34.510,426.031,170.026,33.034,156.233
C01506=1047.666,-34.261,426.018,170.028,33.036,156.234
C01507=1047.673,-34.011,426.004,170.030,33.037,156.234
C01508=1047.679,-33.762,425.991,170.032,33.039,156.234
C01509=1047.686,-33.512,425.978,170.034,33.040,156.234
C01510=1047.692,-33.263,425.964,170.036,33.041,156.234
C01511=1047.698,-33.013,425.952,170.037,33.042,156.234
C01512=1047.704,-32.763,425.938,170.039,33.044,156.235
C01513=1047.710,-32.514,425.924,170.041,33.045,156.235
C01514=1047.716,-32.265,425.911,170.043,33.047,156.235
C01515=1047.723,-32.015,425.897,170.045,33.048,156.235
C01516=1047.729,-31.765,425.884,170.047,33.050,156.235
C01517=1047.735,-31.516,425.871,170.049,33.051,156.235
C01518=1047.742,-31.267,425.858,170.051,33.052,156.236
C01519=1047.748,-31.016,425.845,170.053,33.053,156.236
C01520=1047.754,-30.767,425.831,170.055,33.055,156.236
C01521=1047.761,-30.518,425.818,170.057,33.056,156.236
C01522=1047.767,-30.268,425.805,170.059,33.058,156.236
C01523=1047.773,-30.018,425.791,170.061,33.059,156.236
C01524=1047.779,-29.769,425.777,170.063,33.060,156.237
C01525=1047.786,-29.519,425.764,170.065,33.062,156.237
C01526=1047.792,-29.270,425.751,170.066,33.063,156.237
C01527=1047.798,-29.020,425.737,170.068,33.065,156.237
C01528=1047.805,-28.770,425.724,170.070,33.065,156.237
C01529=1047.811,-28.521,425.710,170.072,33.067,156.237
C01530=1047.818,-28.272,425.697,170.074,33.068,156.238
C01531=1047.824,-28.022,425.683,170.076,33.070,156.238
C01532=1047.830,-27.772,425.670,170.078,33.071,156.238
C01533=1047.836,-27.523,425.656,170.080,33.073,156.238
C01534=1047.843,-27.273,425.643,170.082,33.074,156.238
C01535=1047.849,-27.024,425.629,170.084,33.076,156.239
C01536=1047.856,-26.774,425.616,170.086,33.077,156.239
C01537=1047.861,-26.524,425.602,170.088,33.078,156.239
C01538=1047.868,-26.275,425.589,170.090,33.080,156.239
C01539=1047.874,-26.025,425.575,170.092,33.081,156.239
C01540=1047.880,-25.775,425.561,170.094,33.083,156.240
C01541=1047.886,-25.526,425.548,170.096,33.084,156.240
C01542=1047.892,-25.277,425.533,170.098,33.086,156.240
C01543=1047.899,-25.027,425.520,170.100,33.087,156.240
C01544=1047.905,-24.778,425.506,170.102,33.088,156.240
C01545=1047.911,-24.528,425.492,170.103,33.090,156.241
C01546=1047.917,-24.278,425.479,170.105,33.092,156.241
C01547=1047.923,-24.029,425.466,170.107,33.093,156.241
C01548=1047.930,-23.780,425.451,170.109,33.095,156.241
C01549=1047.936,-23.530,425.437,170.111,33.096,156.241
C01550=1047.942,-23.280,425.423,170.113,33.098,156.241
C01551=1047.948,-23.031,425.410,170.115,33.099,156.242
C01552=1047.955,-22.781,425.397,170.117,33.100,156.242
C01553=1047.961,-22.531,425.382,170.119,33.102,156.242
C01554=1047.967,-22.283,425.368,170.121,33.103,156.242
C01555=1047.973,-22.032,425.354,170.123,33.105,156.242
C01556=1047.979,-21.783,425.341,170.124,33.106,156.243
C01557=1047.986,-21.534,425.328,170.126,33.108,156.243
C01558=1047.992,-21.284,425.313,170.127,33.110,156.243
C01559=1047.998,-21.035,425.299,170.129,33.111,156.243
C01560=1048.005,-20.785,425.286,170.131,33.112,156.243
C01561=1048.010,-20.535,425.272,170.133,33.114,156.244
C01562=1048.018,-20.286,425.258,170.135,33.115,156.244
C01563=1048.023,-20.036,425.244,170.137,33.117,156.244
C01564=1048.030,-19.786,425.230,170.139,33.118,156.244
C01565=1048.036,-19.537,425.215,170.141,33.120,156.244
C01566=1048.043,-19.256,425.201,170.143,33.122,156.245
C01567=1048.051,-18.974,425.185,170.145,33.123,156.245
C01568=1048.057,-18.693,425.169,170.147,33.124,156.245
C01569=1048.064,-18.412,425.153,170.149,33.126,156.245
C01570=1048.070,-18.162,425.139,170.151,33.128,156.246
C01571=1048.077,-17.913,425.125,170.153,33.129,156.246
C01572=1048.083,-17.663,425.111,170.155,33.131,156.246
C01573=1048.089,-17.414,425.098,170.157,33.132,156.246
C01574=1048.096,-17.164,425.083,170.159,33.134,156.246
C01575=1048.102,-16.915,425.070,170.161,33.135,156.247
C01576=1048.109,-16.665,425.055,170.163,33.137,156.247
C01577=1048.115,-16.416,425.041,170.165,33.139,156.247
C01578=1048.121,-16.166,425.028,170.167,33.140,156.247
C01579=1048.128,-15.916,425.013,170.169,33.141,156.247
C01580=1048.134,-15.667,424.999,170.170,33.143,156.248
C01581=1048.140,-15.417,424.985,170.172,33.144,156.248
C01582=1048.147,-15.168,424.971,170.174,33.146,156.248
C01583=1048.153,-14.918,424.956,170.176,33.148,156.248
C01584=1048.159,-14.669,424.943,170.178,33.149,156.248
C01585=1048.165,-14.419,424.929,170.180,33.150,156.249
C01586=1048.171,-14.170,424.914,170.182,33.152,156.249
C01587=1048.178,-13.920,424.901,170.184,33.154,156.249
C01588=1048.184,-13.671,424.886,170.185,33.155,156.249
C01589=1048.190,-13.421,424.871,170.187,33.157,156.249
C01590=1048.196,-13.172,424.858,170.189,33.158,156.250
C01591=1048.203,-12.922,424.843,170.191,33.160,156.250
C01592=1048.209,-12.672,424.829,170.193,33.162,156.250
C01593=1048.215,-12.423,424.815,170.195,33.163,156.250
C01594=1048.221,-12.173,424.800,170.197,33.164,156.251
C01595=1048.227,-11.924,424.786,170.198,33.166,156.251
C01596=1048.234,-11.674,424.772,170.200,33.168,156.251
C01597=1048.240,-11.425,424.758,170.202,33.169,156.251
C01598=1048.246,-11.176,424.743,170.204,33.171,156.252
C01599=1048.252,-10.926,424.729,170.206,33.173,156.252
C01600=1048.259,-10.677,424.714,170.208,33.174,156.252
C01601=1048.265,-10.426,424.700,170.210,33.176,156.252
C01602=1048.270,-10.177,424.686,170.212,33.178,156.252
C01603=1048.278,-9.928,424.671,170.213,33.179,156.253
C01604=1048.283,-9.678,424.657,170.215,33.180,156.253
C01605=1048.289,-9.429,424.642,170.217,33.182,156.253
C01606=1048.297,-9.179,424.628,170.219,33.184,156.253
C01607=1048.302,-8.930,424.614,170.221,33.185,156.253
C01608=1048.308,-8.680,424.599,170.223,33.187,156.254
C01609=1048.316,-8.431,424.585,170.224,33.189,156.254
C01610=1048.321,-8.181,424.571,170.226,33.190,156.254
C01611=1048.327,-7.932,424.556,170.228,33.192,156.254
C01612=1048.334,-7.682,424.541,170.230,33.193,156.255
C01613=1048.340,-7.433,424.528,170.232,33.195,156.255
C01614=1048.346,-7.183,424.513,170.234,33.196,156.255
C01615=1048.353,-6.933,424.498,170.236,33.198,156.255
C01616=1048.359,-6.684,424.483,170.237,33.200,156.256
C01617=1048.365,-6.434,424.470,170.239,33.201,156.256
C01618=1048.372,-6.185,424.455,170.241,33.203,156.256
C01619=1048.378,-5.936,424.440,170.242,33.204,156.256
C01620=1048.385,-5.687,424.426,170.244,33.206,156.256
C01621=1048.391,-5.436,424.412,170.246,33.208,156.257
C01622=1048.396,-5.187,424.397,170.248,33.209,156.257
C01623=1048.403,-4.938,424.382,170.249,33.211,156.257
C01624=1048.410,-4.688,424.368,170.251,33.212,156.257
C01625=1048.416,-4.439,424.353,170.253,33.214,156.257
C01626=1048.422,-4.189,424.339,170.255,33.215,156.258
C01627=1048.428,-3.939,424.324,170.257,33.217,156.258
C01628=1048.435,-3.690,424.310,170.259,33.219,156.258
C01629=1048.441,-3.441,424.295,170.260,33.220,156.258
C01630=1048.448,-3.158,424.279,170.262,33.222,156.259
C01631=1048.456,-2.875,424.262,170.264,33.224,156.259
C01632=1048.462,-2.592,424.244,170.267,33.226,156.259
C01633=1048.469,-2.309,424.228,170.269,33.228,156.260
C01634=1048.475,-2.059,424.213,170.270,33.230,156.260
C01635=1048.481,-1.810,424.198,170.272,33.231,156.260
C01636=1048.487,-1.561,424.184,170.274,33.233,156.260
C01637=1048.494,-1.311,424.169,170.276,33.234,156.260
C01638=1048.500,-1.061,424.154,170.278,33.236,156.261
C01639=1048.506,-0.812,424.139,170.279,33.238,156.261
C01640=1048.512,-0.563,424.124,170.281,33.240,156.261
C01641=1048.519,-0.313,424.109,170.283,33.241,156.261
C01642=1048.525,-0.063,424.094,170.285,33.243,156.262
C01643=1048.531,0.186,424.080,170.287,33.245,156.262
C01644=1048.537,0.435,424.065,170.288,33.247,156.262
C01645=1048.544,0.685,424.050,170.290,33.248,156.262
C01646=1048.549,0.934,424.035,170.292,33.250,156.263
C01647=1048.556,1.184,424.020,170.294,33.252,156.263
C01648=1048.561,1.434,424.005,170.296,33.254,156.263
C01649=1048.568,1.683,423.990,170.297,33.255,156.263
C01650=1048.574,1.932,423.975,170.299,33.257,156.264
C01651=1048.580,2.182,423.960,170.301,33.258,156.264
C01652=1048.586,2.431,423.945,170.303,33.260,156.264
C01653=1048.593,2.681,423.930,170.305,33.262,156.264
C01654=1048.599,2.931,423.915,170.306,33.264,156.265
C01655=1048.605,3.180,423.901,170.308,33.265,156.265
C01656=1048.611,3.429,423.886,170.310,33.267,156.265
C01657=1048.618,3.679,423.871,170.312,33.269,156.265
C01658=1048.624,3.928,423.855,170.313,33.271,156.266
C01659=1048.631,4.178,423.840,170.315,33.272,156.266
C01660=1048.636,4.427,423.826,170.317,33.274,156.266
C01661=1048.642,4.677,423.810,170.319,33.275,156.266
C01662=1048.648,4.926,423.795,170.321,33.277,156.267
C01663=1048.655,5.176,423.780,170.322,33.279,156.267
C01664=1048.661,5.426,423.765,170.324,33.280,156.267
C01665=1048.667,5.674,423.750,170.326,33.282,156.267
C01666=1048.674,5.924,423.735,170.328,33.284,156.268
C01667=1048.680,6.173,423.720,170.330,33.286,156.268
C01668=1048.686,6.423,423.705,170.331,33.287,156.268
C01669=1048.693,6.673,423.690,170.333,33.289,156.268
C01670=1048.700,6.922,423.675,170.335,33.290,156.269
C01671=1048.705,7.172,423.659,170.337,33.292,156.269
C01672=1048.711,7.421,423.645,170.338,33.294,156.269
C01673=1048.717,7.670,423.630,170.340,33.296,156.269
C01674=1048.724,7.920,423.615,170.342,33.297,156.270
C01675=1048.730,8.169,423.599,170.344,33.299,156.270
C01676=1048.737,8.419,423.584,170.346,33.301,156.270
C01677=1048.743,8.668,423.569,170.347,33.303,156.270
C01678=1048.750,8.918,423.554,170.349,33.304,156.271
C01679=1048.756,9.167,423.538,170.351,33.306,156.271
C01680=1048.762,9.417,423.523,170.353,33.308,156.271
C01681=1048.768,9.666,423.508,170.354,33.309,156.271
C01682=1048.774,9.915,423.493,170.356,33.311,156.272
C01683=1048.781,10.165,423.478,170.358,33.313,156.272
C01684=1048.787,10.414,423.463,170.360,33.314,156.272
C01685=1048.794,10.664,423.448,170.361,33.316,156.272
C01686=1048.800,10.913,423.432,170.363,33.318,156.273
C01687=1048.806,11.163,423.417,170.365,33.320,156.273
C01688=1048.812,11.413,423.402,170.367,33.321,156.273
C01689=1048.819,11.662,423.386,170.369,33.323,156.273
C01690=1048.825,11.911,423.371,170.370,33.324,156.274
C01691=1048.832,12.161,423.356,170.372,33.326,156.274
C01692=1048.838,12.410,423.341,170.374,33.328,156.274
C01693=1048.844,12.660,423.325,170.376,33.330,156.274
C01694=1048.851,12.944,423.308,170.378,33.331,156.275
C01695=1048.859,13.229,423.291,170.380,33.333,156.275
C01696=1048.866,13.514,423.273,170.382,33.335,156.275
C01697=1048.874,13.799,423.256,170.384,33.337,156.276
C01698=1048.880,14.048,423.239,170.385,33.339,156.276
C01699=1048.886,14.298,423.224,170.387,33.341,156.276
C01700=1048.892,14.548,423.209,170.389,33.343,156.276
C01701=1048.898,14.797,423.193,170.391,33.344,156.277
C01702=1048.905,15.047,423.178,170.392,33.346,156.277
C01703=1048.911,15.296,423.163,170.394,33.348,156.277
C01704=1048.917,15.546,423.147,170.396,33.350,156.277
C01705=1048.924,15.795,423.131,170.398,33.352,156.278
C01706=1048.929,16.045,423.116,170.399,33.353,156.278
C01707=1048.936,16.294,423.100,170.401,33.355,156.278
C01708=1048.943,16.543,423.085,170.403,33.357,156.279
C01709=1048.948,16.793,423.069,170.405,33.358,156.279
C01710=1048.955,17.042,423.053,170.406,33.360,156.279
C01711=1048.961,17.292,423.038,170.408,33.362,156.279
C01712=1048.967,17.541,423.022,170.410,33.364,156.280
C01713=1048.974,17.790,423.007,170.411,33.366,156.280
C01714=1048.980,18.040,422.991,170.413,33.367,156.280
C01715=1048.986,18.289,422.976,170.415,33.369,156.280
C01716=1048.992,18.539,422.960,170.417,33.371,156.281
C01717=1048.999,18.788,422.944,170.418,33.373,156.281
C01718=1049.005,19.037,422.929,170.420,33.375,156.281
C01719=1049.011,19.287,422.913,170.422,33.376,156.281
C01720=1049.018,19.536,422.898,170.424,33.378,156.282
C01721=1049.024,19.786,422.882,170.425,33.380,156.282
C01722=1049.030,20.035,422.866,170.427,33.381,156.282
C01723=1049.036,20.285,422.850,170.429,33.383,156.283
C01724=1049.043,20.534,422.835,170.430,33.385,156.283
C01725=1049.048,20.783,422.819,170.432,33.387,156.283
C01726=1049.055,21.033,422.804,170.434,33.389,156.283
C01727=1049.061,21.282,422.787,170.436,33.391,156.284
C01728=1049.068,21.531,422.772,170.437,33.392,156.284
C01729=1049.073,21.781,422.756,170.439,33.394,156.284
C01730=1049.079,22.031,422.740,170.441,33.396,156.284
C01731=1049.086,22.280,422.724,170.442,33.397,156.285
C01732=1049.092,22.529,422.708,170.444,33.399,156.285
C01733=1049.098,22.779,422.693,170.446,33.401,156.285
C01734=1049.104,23.028,422.677,170.448,33.403,156.286
C01735=1049.111,23.278,422.661,170.449,33.405,156.286
C01736=1049.117,23.527,422.644,170.451,33.407,156.286
C01737=1049.124,23.777,422.629,170.453,33.409,156.286
C01738=1049.130,24.026,422.613,170.454,33.410,156.287
C01739=1049.136,24.275,422.597,170.456,33.412,156.287
C01740=1049.142,24.524,422.581,170.458,33.414,156.287
C01741=1049.148,24.774,422.565,170.460,33.416,156.287
C01742=1049.155,25.023,422.550,170.461,33.418,156.288
C01743=1049.161,25.273,422.534,170.463,33.420,156.288
C01744=1049.167,25.522,422.518,170.465,33.421,156.288
C01745=1049.174,25.772,422.502,170.466,33.423,156.289
C01746=1049.179,25.995,422.487,170.468,33.424,156.289
C01747=1049.185,26.219,422.473,170.469,33.426,156.289
C01748=1049.190,26.442,422.459,170.471,33.428,156.289
C01749=1049.196,26.665,422.444,170.473,33.430,156.290
C01750=1049.201,26.889,422.430,170.474,33.431,156.290
C01751=1049.207,27.112,422.417,170.476,33.433,156.290
C01752=1049.213,27.336,422.402,170.477,33.434,156.290
C01753=1049.219,27.559,422.387,170.479,33.436,156.291
C01754=1049.225,27.809,422.371,170.480,33.438,156.291
C01755=1049.231,28.058,422.355,170.482,33.440,156.291
C01756=1049.237,28.307,422.339,170.484,33.441,156.291
C01757=1049.243,28.556,422.323,170.485,33.443,156.292
C01758=1049.252,28.895,422.301,170.488,33.446,156.292
C01759=1049.261,29.233,422.279,170.490,33.448,156.293
C01760=1049.269,29.572,422.257,170.492,33.451,156.293
C01761=1049.277,29.909,422.236,170.495,33.453,156.293
C01762=1049.283,30.158,422.219,170.496,33.455,156.294
C01763=1049.290,30.408,422.203,170.498,33.457,156.294
C01764=1049.296,30.658,422.187,170.500,33.459,156.294
C01765=1049.302,30.907,422.170,170.501,33.460,156.294
C01766=1049.308,31.156,422.155,170.503,33.462,156.295
C01767=1049.314,31.405,422.138,170.505,33.464,156.295
C01768=1049.321,31.656,422.122,170.506,33.466,156.295
C01769=1049.327,31.905,422.106,170.508,33.468,156.296
C01770=1049.333,32.154,422.089,170.510,33.470,156.296
C01771=1049.339,32.403,422.074,170.511,33.472,156.296
C01772=1049.345,32.653,422.057,170.513,33.474,156.296
C01773=1049.351,32.902,422.041,170.515,33.476,156.297
C01774=1049.358,33.152,422.024,170.516,33.477,156.297
C01775=1049.364,33.401,422.008,170.518,33.479,156.297
C01776=1049.371,33.650,421.992,170.521,33.481,156.298
C01777=1049.377,33.899,421.976,170.522,33.483,156.298
C01778=1049.383,34.149,421.959,170.524,33.485,156.298
C01779=1049.389,34.399,421.943,170.526,33.486,156.298
C01780=1049.395,34.648,421.926,170.528,33.488,156.299
C01781=1049.401,34.897,421.910,170.529,33.490,156.299
C01782=1049.408,35.147,421.894,170.531,33.492,156.299
C01783=1049.414,35.396,421.878,170.533,33.494,156.300
C01784=1049.421,35.645,421.861,170.534,33.496,156.300
C01785=1049.427,35.894,421.845,170.536,33.498,156.300
C01786=1049.433,36.144,421.828,170.538,33.500,156.300
C01787=1049.439,36.394,421.812,170.539,33.501,156.301
C01788=1049.446,36.643,421.796,170.541,33.503,156.301
C01789=1049.452,36.892,421.779,170.543,33.505,156.301
C01790=1049.459,37.142,421.763,170.544,33.507,156.302
C01791=1049.465,37.391,421.746,170.546,33.509,156.302
C01792=1049.470,37.640,421.730,170.548,33.510,156.302
C01793=1049.477,37.890,421.713,170.549,33.512,156.302
C01794=1049.483,38.139,421.696,170.551,33.514,156.303
C01795=1049.489,38.388,421.680,170.553,33.516,156.303
C01796=1049.495,38.638,421.664,170.554,33.518,156.303
C01797=1049.502,38.888,421.647,170.556,33.520,156.304
C01798=1049.508,39.137,421.630,170.558,33.522,156.304
C01799=1049.514,39.386,421.614,170.559,33.524,156.304
C01800=1049.520,39.635,421.598,170.561,33.526,156.305
C01801=1049.527,39.885,421.580,170.563,33.528,156.305
C01802=1049.533,40.134,421.564,170.564,33.530,156.305
C01803=1049.539,40.383,421.548,170.566,33.532,156.306
C01804=1049.545,40.633,421.531,170.568,33.534,156.306
C01805=1049.551,40.882,421.514,170.569,33.536,156.306
C01806=1049.557,41.132,421.498,170.571,33.537,156.306
C01807=1049.564,41.381,421.480,170.573,33.539,156.307
C01808=1049.569,41.631,421.464,170.574,33.541,156.307
C01809=1049.576,41.879,421.447,170.576,33.543,156.307
C01810=1049.582,42.129,421.430,170.577,33.545,156.308
C01811=1049.588,42.379,421.414,170.579,33.547,156.308
C01812=1049.594,42.627,421.397,170.581,33.549,156.308
C01813=1049.601,42.878,421.380,170.582,33.550,156.308
C01814=1049.607,43.127,421.364,170.584,33.552,156.309
C01815=1049.613,43.376,421.347,170.586,33.554,156.309
C01816=1049.620,43.626,421.331,170.587,33.556,156.309
C01817=1049.625,43.875,421.313,170.589,33.558,156.310
C01818=1049.631,44.124,421.297,170.591,33.560,156.310
